LIN {X 0,Y 361.952,Z 273.021,A -85,B 0,C 180,E1 -12972.333,E2 -12972.333} C_VEL
LIN {X 0,Y 361.954,Z 273.018,A -85,B 0,C 180,E1 -12974.621,E2 -12974.621} C_VEL
LIN {X 0,Y 361.95,Z 273.019,A -85,B 0,C 180,E1 -12978.1,E2 -12978.1} C_VEL
LIN {X 0,Y 361.885,Z 273.022,A -85,B 0,C 180,E1 -12981.653,E2 -12981.653} C_VEL
LIN {X 0,Y 361.922,Z 273.026,A -85,B 0,C 180,E1 -12985.29,E2 -12985.29} C_VEL
LIN {X 0,Y 361.916,Z 273.017,A -85,B 0,C 180,E1 -12987.778,E2 -12987.778} C_VEL
LIN {X 0,Y 361.841,Z 273.035,A -85,B 0,C 180,E1 -12991.286,E2 -12991.286} C_VEL
LIN {X 0,Y 361.849,Z 272.995,A -85,B 0,C 180,E1 -12994.281,E2 -12994.281} C_VEL
LIN {X 0,Y 361.86,Z 273.028,A -85,B 0,C 180,E1 -12997.224,E2 -12997.224} C_VEL
LIN {X 0,Y 361.831,Z 273.03,A -85,B 0,C 180,E1 -13000.756,E2 -13000.756} C_VEL
LIN {X 0,Y 361.842,Z 273.033,A -85,B 0,C 180,E1 -13004.365,E2 -13004.365} C_VEL
LIN {X 0,Y 361.88,Z 273.014,A -85,B 0,C 180,E1 -13007.561,E2 -13007.561} C_VEL
LIN {X 0,Y 361.872,Z 273.035,A -85,B 0,C 180,E1 -13010.973,E2 -13010.973} C_VEL
LIN {X 0,Y 361.872,Z 273.035,A -85,B 0,C 180,E1 -13014.656,E2 -13014.656} C_VEL
LIN {X 0,Y 361.866,Z 273.12,A -85,B 0,C 180,E1 -13017.718,E2 -13017.718} C_VEL
LIN {X 0,Y 364.625,Z 284.445,A -85,B 0,C 180,E1 -13020.757,E2 -13020.757} C_VEL
LIN {X 0,Y 366.783,Z 294.302,A -85,B 0,C 180,E1 -13023.166,E2 -13023.166} C_VEL
LIN {X 0,Y 369.556,Z 302.023,A -85,B 0,C 180,E1 -13023.576,E2 -13023.576} C_VEL
LIN {X 0,Y 374.934,Z 329.513,A -85,B 0,C 180,E1 -13024.555,E2 -13024.555} C_VEL
LIN {X 0,Y 373.046,Z 425.138,A -85,B 0,C 180,E1 -13026.401,E2 -13026.401} C_VEL
LIN {X 0,Y 372.477,Z 438.942,A -85,B 0,C 180,E1 -13026.768,E2 -13026.768} C_VEL
LIN {X 0,Y 371.561,Z 452.604,A -85,B 0,C 180,E1 -13027.333,E2 -13027.333} C_VEL
LIN {X 0,Y 370.455,Z 465.982,A -85,B 0,C 180,E1 -13028.106,E2 -13028.106} C_VEL
LIN {X 0,Y 369.2,Z 479.198,A -85,B 0,C 180,E1 -13029.112,E2 -13029.112} C_VEL
LIN {X 0,Y 367.718,Z 491.74,A -85,B 0,C 180,E1 -13030.315,E2 -13030.315} C_VEL
LIN {X 0,Y 366.376,Z 502.198,A -85,B 0,C 180,E1 -13031.548,E2 -13031.548} C_VEL
LIN {X 0,Y 365.092,Z 511.93,A -85,B 0,C 180,E1 -13032.929,E2 -13032.929} C_VEL
LIN {X 0,Y 363.782,Z 521.814,A -85,B 0,C 180,E1 -13034.624,E2 -13034.624} C_VEL
LIN {X 0,Y 362.74,Z 529.741,A -85,B 0,C 180,E1 -13036.271,E2 -13036.271} C_VEL
LIN {X 0,Y 361.767,Z 537.481,A -85,B 0,C 180,E1 -13038.23,E2 -13038.23} C_VEL
LIN {X 0,Y 361.155,Z 542.884,A -85,B 0,C 180,E1 -13039.914,E2 -13039.914} C_VEL
LIN {X 0,Y 360.659,Z 548.569,A -85,B 0,C 180,E1 -13042.16,E2 -13042.16} C_VEL
LIN {X 0,Y 360.407,Z 552.693,A -85,B 0,C 180,E1 -13044.405,E2 -13044.405} C_VEL
LIN {X 0,Y 360.267,Z 555.385,A -85,B 0,C 180,E1 -13046.645,E2 -13046.645} C_VEL
LIN {X 0,Y 360.246,Z 556.718,A -85,B 0,C 180,E1 -13048.882,E2 -13048.882} C_VEL
LIN {X 0,Y 360.246,Z 556.714,A -85,B 0,C 180,E1 -13051.118,E2 -13051.118} C_VEL
LIN {X 0,Y 360.268,Z 555.376,A -85,B 0,C 180,E1 -13053.355,E2 -13053.355} C_VEL
LIN {X 0,Y 360.408,Z 552.678,A -85,B 0,C 180,E1 -13055.595,E2 -13055.595} C_VEL
LIN {X 0,Y 360.659,Z 548.543,A -85,B 0,C 180,E1 -13057.84,E2 -13057.84} C_VEL
LIN {X 0,Y 361.163,Z 542.848,A -85,B 0,C 180,E1 -13060.086,E2 -13060.086} C_VEL
LIN {X 0,Y 361.932,Z 536.429,A -85,B 0,C 180,E1 -13062.049,E2 -13062.049} C_VEL
LIN {X 0,Y 362.885,Z 528.492,A -85,B 0,C 180,E1 -13064.001,E2 -13064.001} C_VEL
LIN {X 0,Y 363.958,Z 520.11,A -85,B 0,C 180,E1 -13065.684,E2 -13065.684} C_VEL
LIN {X 0,Y 365.283,Z 510.065,A -85,B 0,C 180,E1 -13067.35,E2 -13067.35} C_VEL
LIN {X 0,Y 366.763,Z 498.857,A -85,B 0,C 180,E1 -13068.866,E2 -13068.866} C_VEL
LIN {X 0,Y 368.224,Z 487.708,A -85,B 0,C 180,E1 -13070.093,E2 -13070.093} C_VEL
LIN {X 0,Y 369.54,Z 475.56,A -85,B 0,C 180,E1 -13071.182,E2 -13071.182} C_VEL
LIN {X 0,Y 370.771,Z 462.078,A -85,B 0,C 180,E1 -13072.131,E2 -13072.131} C_VEL
LIN {X 0,Y 371.888,Z 447.972,A -85,B 0,C 180,E1 -13072.867,E2 -13072.867} C_VEL
LIN {X 0,Y 372.638,Z 434.166,A -85,B 0,C 180,E1 -13073.369,E2 -13073.369} C_VEL
LIN {X 0,Y 373.32,Z 411.975,A -85,B 0,C 180,E1 -13073.838,E2 -13073.838} C_VEL
LIN {X 0,Y 374.849,Z 329.127,A -85,B 0,C 180,E1 -13075.444,E2 -13075.444} C_VEL
LIN {X 0,Y 369.224,Z 300.604,A -85,B 0,C 180,E1 -13076.464,E2 -13076.464} C_VEL
LIN {X 0,Y 366.745,Z 294.208,A -85,B 0,C 180,E1 -13076.829,E2 -13076.829} C_VEL
LIN {X 0,Y 364.591,Z 284.391,A -85,B 0,C 180,E1 -13079.241,E2 -13079.241} C_VEL
LIN {X 0,Y 361.892,Z 273.253,A -85,B 0,C 180,E1 -13082.197,E2 -13082.197} C_VEL
LIN {X 0,Y 361.852,Z 273.028,A -85,B 0,C 180,E1 -13084.28,E2 -13084.28} C_VEL
LIN {X 0,Y 361.861,Z 273.02,A -85,B 0,C 180,E1 -13087.222,E2 -13087.222} C_VEL
LIN {X 0,Y 361.832,Z 273.02,A -85,B 0,C 180,E1 -13090.755,E2 -13090.755} C_VEL
LIN {X 0,Y 361.816,Z 273.043,A -85,B 0,C 180,E1 -13094.368,E2 -13094.368} C_VEL
LIN {X 0,Y 361.833,Z 273.038,A -85,B 0,C 180,E1 -13097.567,E2 -13097.567} C_VEL
LIN {X 0,Y 361.867,Z 273.034,A -85,B 0,C 180,E1 -13100.973,E2 -13100.973} C_VEL
LIN {X 0,Y 361.87,Z 272.997,A -85,B 0,C 180,E1 -13104.655,E2 -13104.655} C_VEL
LIN {X 0,Y 361.833,Z 273.03,A -85,B 0,C 180,E1 -13108.37,E2 -13108.37} C_VEL
LIN {X 0,Y 361.897,Z 273.027,A -85,B 0,C 180,E1 -13110.955,E2 -13110.955} C_VEL
LIN {X 0,Y 361.949,Z 273.015,A -85,B 0,C 180,E1 -13113.475,E2 -13113.475} C_VEL
LIN {X 0,Y 361.884,Z 273.023,A -85,B 0,C 180,E1 -13117.144,E2 -13117.144} C_VEL
LIN {X 0,Y 361.905,Z 273.028,A -85,B 0,C 180,E1 -13120.723,E2 -13120.723} C_VEL
LIN {X 0,Y 361.926,Z 273.015,A -85,B 0,C 180,E1 -13123.066,E2 -13123.066} C_VEL
LIN {X 0,Y 361.992,Z 273.017,A -85,B 0,C 180,E1 -13126.528,E2 -13126.528} C_VEL
LIN {X 0,Y 362.024,Z 273.001,A -85,B 0,C 180,E1 -13129.938,E2 -13129.938} C_VEL
LIN {X 0,Y 362.144,Z 272.999,A -85,B 0,C 180,E1 -13132.192,E2 -13132.192} C_VEL
LIN {X 0,Y 362.111,Z 272.996,A -85,B 0,C 180,E1 -13134.431,E2 -13134.431} C_VEL
LIN {X 0,Y 362.275,Z 272.979,A -85,B 0,C 180,E1 -13137.776,E2 -13137.776} C_VEL
LIN {X 0,Y 362.42,Z 272.962,A -85,B 0,C 180,E1 -13140,E2 -13140} C_VEL
LIN {X 0,Y 362.276,Z 272.964,A -85,B 0,C 180,E1 -13142.224,E2 -13142.224} C_VEL
LIN {X 0,Y 362.156,Z 272.996,A -85,B 0,C 180,E1 -13146.687,E2 -13146.687} C_VEL
LIN {X 0,Y 362.024,Z 273.008,A -85,B 0,C 180,E1 -13150.062,E2 -13150.062} C_VEL
LIN {X 0,Y 361.991,Z 273.008,A -85,B 0,C 180,E1 -13153.899,E2 -13153.899} C_VEL
LIN {X 0,Y 361.961,Z 273.021,A -85,B 0,C 180,E1 -13157.939,E2 -13157.939} C_VEL
LIN {X 0,Y 361.886,Z 273.024,A -85,B 0,C 180,E1 -13161.653,E2 -13161.653} C_VEL
LIN {X 0,Y 361.923,Z 273.018,A -85,B 0,C 180,E1 -13165.291,E2 -13165.291} C_VEL
LIN {X 0,Y 361.917,Z 273.025,A -85,B 0,C 180,E1 -13167.778,E2 -13167.778} C_VEL
LIN {X 0,Y 361.842,Z 273.019,A -85,B 0,C 180,E1 -13171.286,E2 -13171.286} C_VEL
LIN {X 0,Y 361.85,Z 272.997,A -85,B 0,C 180,E1 -13174.281,E2 -13174.281} C_VEL
LIN {X 0,Y 361.868,Z 273.036,A -85,B 0,C 180,E1 -13177.225,E2 -13177.225} C_VEL
LIN {X 0,Y 361.852,Z 273.006,A -85,B 0,C 180,E1 -13180.76,E2 -13180.76} C_VEL
LIN {X 0,Y 361.832,Z 273.037,A -85,B 0,C 180,E1 -13184.367,E2 -13184.367} C_VEL
LIN {X 0,Y 361.834,Z 273.015,A -85,B 0,C 180,E1 -13187.569,E2 -13187.569} C_VEL
LIN {X 0,Y 361.868,Z 273.03,A -85,B 0,C 180,E1 -13190.974,E2 -13190.974} C_VEL
LIN {X 0,Y 361.873,Z 273.032,A -85,B 0,C 180,E1 -13194.656,E2 -13194.656} C_VEL
LIN {X 0,Y 361.837,Z 273.032,A -85,B 0,C 180,E1 -13198.371,E2 -13198.371} C_VEL
LIN {X 0,Y 361.901,Z 273.139,A -85,B 0,C 180,E1 -13199.064,E2 -13199.064} C_VEL
LIN {X 0,Y 364.583,Z 284.299,A -85,B 0,C 180,E1 -13202.131,E2 -13202.131} C_VEL
LIN {X 0,Y 365.464,Z 288.404,A -85,B 0,C 180,E1 -13203.13,E2 -13203.13} C_VEL
LIN {X 0,Y 371.55,Z 303.667,A -85,B 0,C 180,E1 -13203.956,E2 -13203.956} C_VEL
LIN {X 0,Y 375.122,Z 322.173,A -85,B 0,C 180,E1 -13204.608,E2 -13204.608} C_VEL
LIN {X 0,Y 373.223,Z 410.537,A -85,B 0,C 180,E1 -13206.303,E2 -13206.303} C_VEL
LIN {X 0,Y 372.705,Z 428.632,A -85,B 0,C 180,E1 -13206.709,E2 -13206.709} C_VEL
LIN {X 0,Y 371.91,Z 442.893,A -85,B 0,C 180,E1 -13207.245,E2 -13207.245} C_VEL
LIN {X 0,Y 370.856,Z 457.001,A -85,B 0,C 180,E1 -13208.008,E2 -13208.008} C_VEL
LIN {X 0,Y 369.689,Z 470.266,A -85,B 0,C 180,E1 -13208.972,E2 -13208.972} C_VEL
LIN {X 0,Y 368.352,Z 482.146,A -85,B 0,C 180,E1 -13210.06,E2 -13210.06} C_VEL
LIN {X 0,Y 366.843,Z 494.177,A -85,B 0,C 180,E1 -13211.428,E2 -13211.428} C_VEL
LIN {X 0,Y 365.427,Z 505.023,A -85,B 0,C 180,E1 -13212.945,E2 -13212.945} C_VEL
LIN {X 0,Y 363.998,Z 515.188,A -85,B 0,C 180,E1 -13214.683,E2 -13214.683} C_VEL
LIN {X 0,Y 362.971,Z 524.109,A -85,B 0,C 180,E1 -13216.565,E2 -13216.565} C_VEL
LIN {X 0,Y 362.003,Z 530.634,A -85,B 0,C 180,E1 -13218.238,E2 -13218.238} C_VEL
LIN {X 0,Y 361.393,Z 536.049,A -85,B 0,C 180,E1 -13219.92,E2 -13219.92} C_VEL
LIN {X 0,Y 360.776,Z 541.742,A -85,B 0,C 180,E1 -13222.163,E2 -13222.163} C_VEL
LIN {X 0,Y 360.623,Z 544.719,A -85,B 0,C 180,E1 -13223.677,E2 -13223.677} C_VEL
LIN {X 0,Y 360.423,Z 547.405,A -85,B 0,C 180,E1 -13225.527,E2 -13225.527} C_VEL
LIN {X 0,Y 360.263,Z 549.43,A -85,B 0,C 180,E1 -13227.764,E2 -13227.764} C_VEL
LIN {X 0,Y 360.274,Z 550.124,A -85,B 0,C 180,E1 -13230,E2 -13230} C_VEL
LIN {X 0,Y 360.263,Z 549.497,A -85,B 0,C 180,E1 -13232.236,E2 -13232.236} C_VEL
LIN {X 0,Y 360.423,Z 547.532,A -85,B 0,C 180,E1 -13234.473,E2 -13234.473} C_VEL
LIN {X 0,Y 360.655,Z 544.185,A -85,B 0,C 180,E1 -13236.714,E2 -13236.714} C_VEL
LIN {X 0,Y 361.032,Z 539.358,A -85,B 0,C 180,E1 -13238.959,E2 -13238.959} C_VEL
LIN {X 0,Y 361.73,Z 532.895,A -85,B 0,C 180,E1 -13241.203,E2 -13241.203} C_VEL
LIN {X 0,Y 362.715,Z 525.696,A -85,B 0,C 180,E1 -13243.159,E2 -13243.159} C_VEL
LIN {X 0,Y 363.758,Z 517.473,A -85,B 0,C 180,E1 -13244.977,E2 -13244.977} C_VEL
LIN {X 0,Y 364.828,Z 509.096,A -85,B 0,C 180,E1 -13246.507,E2 -13246.507} C_VEL
LIN {X 0,Y 366.341,Z 498.123,A -85,B 0,C 180,E1 -13248.164,E2 -13248.164} C_VEL
LIN {X 0,Y 367.661,Z 488.275,A -85,B 0,C 180,E1 -13249.38,E2 -13249.38} C_VEL
LIN {X 0,Y 367.626,Z 483.577,A -85,B 0,C 180,E1 -13249.941,E2 -13249.941} C_VEL
LIN {X 0,Y 365.814,Z 475.828,A -85,B 0,C 180,E1 -13250.871,E2 -13250.871} C_VEL
LIN {X 0,Y 363.955,Z 467.722,A -85,B 0,C 180,E1 -13251.719,E2 -13251.719} C_VEL
LIN {X 0,Y 363.828,Z 462.47,A -85,B 0,C 180,E1 -13252.144,E2 -13252.144} C_VEL
LIN {X 0,Y 365.032,Z 448.328,A -85,B 0,C 180,E1 -13253.021,E2 -13253.021} C_VEL
LIN {X 0,Y 365.932,Z 434.613,A -85,B 0,C 180,E1 -13253.635,E2 -13253.635} C_VEL
LIN {X 0,Y 366.616,Z 420.613,A -85,B 0,C 180,E1 -13254.038,E2 -13254.038} C_VEL
LIN {X 0,Y 368.716,Z 323.276,A -85,B 0,C 180,E1 -13255.95,E2 -13255.95} C_VEL
LIN {X 0,Y 365.307,Z 305.617,A -85,B 0,C 180,E1 -13256.591,E2 -13256.591} C_VEL
LIN {X 0,Y 358.198,Z 288.358,A -85,B 0,C 180,E1 -13257.582,E2 -13257.582} C_VEL
LIN {X 0,Y 355.906,Z 278.366,A -85,B 0,C 180,E1 -13260.247,E2 -13260.247} C_VEL
LIN {X 0,Y 354.815,Z 273.973,A -85,B 0,C 180,E1 -13261.57,E2 -13261.57} C_VEL
LIN {X 0,Y 354.81,Z 273.909,A -85,B 0,C 180,E1 -13265.058,E2 -13265.058} C_VEL
LIN {X 0,Y 354.804,Z 273.901,A -85,B 0,C 180,E1 -13267.882,E2 -13267.882} C_VEL
LIN {X 0,Y 354.786,Z 273.905,A -85,B 0,C 180,E1 -13271.171,E2 -13271.171} C_VEL
LIN {X 0,Y 354.787,Z 273.914,A -85,B 0,C 180,E1 -13274.51,E2 -13274.51} C_VEL
LIN {X 0,Y 354.796,Z 273.888,A -85,B 0,C 180,E1 -13277.663,E2 -13277.663} C_VEL
LIN {X 0,Y 354.815,Z 273.904,A -85,B 0,C 180,E1 -13280.666,E2 -13280.666} C_VEL
LIN {X 0,Y 354.817,Z 273.902,A -85,B 0,C 180,E1 -13284.3,E2 -13284.3} C_VEL
LIN {X 0,Y 354.782,Z 273.881,A -85,B 0,C 180,E1 -13287.666,E2 -13287.666} C_VEL
LIN {X 0,Y 354.863,Z 273.906,A -85,B 0,C 180,E1 -13290.621,E2 -13290.621} C_VEL
LIN {X 0,Y 354.893,Z 273.89,A -85,B 0,C 180,E1 -13294.172,E2 -13294.172} C_VEL
LIN {X 0,Y 354.828,Z 273.905,A -85,B 0,C 180,E1 -13297.893,E2 -13297.893} C_VEL
LIN {X 0,Y 354.916,Z 273.898,A -85,B 0,C 180,E1 -13301.891,E2 -13301.891} C_VEL
LIN {X 0,Y 354.935,Z 273.886,A -85,B 0,C 180,E1 -13305.981,E2 -13305.981} C_VEL
LIN {X 0,Y 354.971,Z 273.886,A -85,B 0,C 180,E1 -13309.736,E2 -13309.736} C_VEL
LIN {X 0,Y 355.12,Z 273.873,A -85,B 0,C 180,E1 -13313.18,E2 -13313.18} C_VEL
LIN {X 0,Y 355.238,Z 273.84,A -85,B 0,C 180,E1 -13317.732,E2 -13317.732} C_VEL
LIN {X 0,Y 355.391,Z 273.837,A -85,B 0,C 180,E1 -13320,E2 -13320} C_VEL
LIN {X 0,Y 355.238,Z 273.855,A -85,B 0,C 180,E1 -13322.268,E2 -13322.268} C_VEL
LIN {X 0,Y 355.13,Z 273.873,A -85,B 0,C 180,E1 -13326.819,E2 -13326.819} C_VEL
LIN {X 0,Y 355.007,Z 273.878,A -85,B 0,C 180,E1 -13329.112,E2 -13329.112} C_VEL
LIN {X 0,Y 354.913,Z 273.901,A -85,B 0,C 180,E1 -13332.581,E2 -13332.581} C_VEL
LIN {X 0,Y 354.882,Z 273.891,A -85,B 0,C 180,E1 -13336.096,E2 -13336.096} C_VEL
LIN {X 0,Y 354.896,Z 273.903,A -85,B 0,C 180,E1 -13338.472,E2 -13338.472} C_VEL
LIN {X 0,Y 354.828,Z 273.899,A -85,B 0,C 180,E1 -13342.106,E2 -13342.106} C_VEL
LIN {X 0,Y 354.893,Z 273.901,A -85,B 0,C 180,E1 -13345.828,E2 -13345.828} C_VEL
LIN {X 0,Y 354.848,Z 273.909,A -85,B 0,C 180,E1 -13349.679,E2 -13349.679} C_VEL
LIN {X 0,Y 354.801,Z 273.875,A -85,B 0,C 180,E1 -13353.703,E2 -13353.703} C_VEL
LIN {X 0,Y 354.793,Z 273.896,A -85,B 0,C 180,E1 -13356.46,E2 -13356.46} C_VEL
LIN {X 0,Y 354.819,Z 273.911,A -85,B 0,C 180,E1 -13359.424,E2 -13359.424} C_VEL
LIN {X 0,Y 354.786,Z 273.915,A -85,B 0,C 180,E1 -13362.868,E2 -13362.868} C_VEL
LIN {X 0,Y 354.837,Z 273.908,A -85,B 0,C 180,E1 -13366.116,E2 -13366.116} C_VEL
LIN {X 0,Y 354.853,Z 273.889,A -85,B 0,C 180,E1 -13369.189,E2 -13369.189} C_VEL
LIN {X 0,Y 354.806,Z 273.899,A -85,B 0,C 180,E1 -13372.403,E2 -13372.403} C_VEL
LIN {X 0,Y 354.81,Z 273.915,A -85,B 0,C 180,E1 -13374.942,E2 -13374.942} C_VEL
LIN {X 0,Y 354.846,Z 274.024,A -85,B 0,C 180,E1 -13377.253,E2 -13377.253} C_VEL
LIN {X 0,Y 357.781,Z 286.229,A -85,B 0,C 180,E1 -13380.589,E2 -13380.589} C_VEL
LIN {X 0,Y 359.57,Z 294.104,A -85,B 0,C 180,E1 -13382.57,E2 -13382.57} C_VEL
LIN {X 0,Y 363.378,Z 304.123,A -85,B 0,C 180,E1 -13383.137,E2 -13383.137} C_VEL
LIN {X 0,Y 368.52,Z 330.505,A -85,B 0,C 180,E1 -13384.102,E2 -13384.102} C_VEL
LIN {X 0,Y 366.561,Z 425.089,A -85,B 0,C 180,E1 -13385.958,E2 -13385.958} C_VEL
LIN {X 0,Y 365.955,Z 438.886,A -85,B 0,C 180,E1 -13386.329,E2 -13386.329} C_VEL
LIN {X 0,Y 365.028,Z 452.545,A -85,B 0,C 180,E1 -13386.904,E2 -13386.904} C_VEL
LIN {X 0,Y 363.867,Z 465.921,A -85,B 0,C 180,E1 -13387.688,E2 -13387.688} C_VEL
LIN {X 0,Y 362.68,Z 477.912,A -85,B 0,C 180,E1 -13388.603,E2 -13388.603} C_VEL
LIN {X 0,Y 361.209,Z 490.384,A -85,B 0,C 180,E1 -13389.797,E2 -13389.797} C_VEL
LIN {X 0,Y 359.588,Z 502.134,A -85,B 0,C 180,E1 -13391.187,E2 -13391.187} C_VEL
LIN {X 0,Y 358.278,Z 511.866,A -85,B 0,C 180,E1 -13392.594,E2 -13392.594} C_VEL
LIN {X 0,Y 356.897,Z 521.749,A -85,B 0,C 180,E1 -13394.32,E2 -13394.32} C_VEL
LIN {X 0,Y 355.646,Z 530.909,A -85,B 0,C 180,E1 -13396.283,E2 -13396.283} C_VEL
LIN {X 0,Y 354.798,Z 537.416,A -85,B 0,C 180,E1 -13397.996,E2 -13397.996} C_VEL
LIN {X 0,Y 354.138,Z 542.818,A -85,B 0,C 180,E1 -13399.712,E2 -13399.712} C_VEL
LIN {X 0,Y 353.602,Z 548.503,A -85,B 0,C 180,E1 -13402.003,E2 -13402.003} C_VEL
LIN {X 0,Y 353.329,Z 552.627,A -85,B 0,C 180,E1 -13404.292,E2 -13404.292} C_VEL
LIN {X 0,Y 353.191,Z 555.319,A -85,B 0,C 180,E1 -13406.578,E2 -13406.578} C_VEL
LIN {X 0,Y 353.146,Z 556.651,A -85,B 0,C 180,E1 -13408.86,E2 -13408.86} C_VEL
LIN {X 0,Y 353.146,Z 556.648,A -85,B 0,C 180,E1 -13411.14,E2 -13411.14} C_VEL
LIN {X 0,Y 353.191,Z 555.31,A -85,B 0,C 180,E1 -13413.422,E2 -13413.422} C_VEL
LIN {X 0,Y 353.329,Z 552.611,A -85,B 0,C 180,E1 -13415.708,E2 -13415.708} C_VEL
LIN {X 0,Y 353.602,Z 548.475,A -85,B 0,C 180,E1 -13417.997,E2 -13417.997} C_VEL
LIN {X 0,Y 354.144,Z 542.78,A -85,B 0,C 180,E1 -13420.288,E2 -13420.288} C_VEL
LIN {X 0,Y 354.96,Z 536.361,A -85,B 0,C 180,E1 -13422.289,E2 -13422.289} C_VEL
LIN {X 0,Y 355.924,Z 528.696,A -85,B 0,C 180,E1 -13424.216,E2 -13424.216} C_VEL
LIN {X 0,Y 357.072,Z 520.041,A -85,B 0,C 180,E1 -13425.995,E2 -13425.995} C_VEL
LIN {X 0,Y 358.484,Z 509.996,A -85,B 0,C 180,E1 -13427.69,E2 -13427.69} C_VEL
LIN {X 0,Y 360.048,Z 498.787,A -85,B 0,C 180,E1 -13429.232,E2 -13429.232} C_VEL
LIN {X 0,Y 361.704,Z 486.351,A -85,B 0,C 180,E1 -13430.605,E2 -13430.605} C_VEL
LIN {X 0,Y 363.131,Z 473.38,A -85,B 0,C 180,E1 -13431.753,E2 -13431.753} C_VEL
LIN {X 0,Y 364.32,Z 460.986,A -85,B 0,C 180,E1 -13432.612,E2 -13432.612} C_VEL
LIN {X 0,Y 365.423,Z 447.135,A -85,B 0,C 180,E1 -13433.332,E2 -13433.332} C_VEL
LIN {X 0,Y 366.189,Z 432.947,A -85,B 0,C 180,E1 -13433.843,E2 -13433.843} C_VEL
LIN {X 0,Y 367.019,Z 402.941,A -85,B 0,C 180,E1 -13434.462,E2 -13434.462} C_VEL
LIN {X 0,Y 368.44,Z 330.261,A -85,B 0,C 180,E1 -13435.894,E2 -13435.894} C_VEL
LIN {X 0,Y 363.186,Z 303.268,A -85,B 0,C 180,E1 -13436.879,E2 -13436.879} C_VEL
LIN {X 0,Y 359.527,Z 294.085,A -85,B 0,C 180,E1 -13437.418,E2 -13437.418} C_VEL
LIN {X 0,Y 356.951,Z 282.742,A -85,B 0,C 180,E1 -13440.312,E2 -13440.312} C_VEL
LIN {X 0,Y 354.846,Z 273.997,A -85,B 0,C 180,E1 -13442.747,E2 -13442.747} C_VEL
LIN {X 0,Y 354.795,Z 273.902,A -85,B 0,C 180,E1 -13446.459,E2 -13446.459} C_VEL
LIN {X 0,Y 354.821,Z 273.912,A -85,B 0,C 180,E1 -13449.423,E2 -13449.423} C_VEL
LIN {X 0,Y 354.785,Z 273.904,A -85,B 0,C 180,E1 -13452.867,E2 -13452.867} C_VEL
LIN {X 0,Y 354.764,Z 273.914,A -85,B 0,C 180,E1 -13456.103,E2 -13456.103} C_VEL
LIN {X 0,Y 354.784,Z 273.907,A -85,B 0,C 180,E1 -13459.178,E2 -13459.178} C_VEL
LIN {X 0,Y 354.804,Z 273.909,A -85,B 0,C 180,E1 -13462.402,E2 -13462.402} C_VEL
LIN {X 0,Y 354.807,Z 273.872,A -85,B 0,C 180,E1 -13464.94,E2 -13464.94} C_VEL
LIN {X 0,Y 354.789,Z 273.907,A -85,B 0,C 180,E1 -13468.404,E2 -13468.404} C_VEL
LIN {X 0,Y 354.848,Z 273.902,A -85,B 0,C 180,E1 -13471.619,E2 -13471.619} C_VEL
LIN {X 0,Y 354.894,Z 273.902,A -85,B 0,C 180,E1 -13474.172,E2 -13474.172} C_VEL
LIN {X 0,Y 354.828,Z 273.899,A -85,B 0,C 180,E1 -13477.894,E2 -13477.894} C_VEL
LIN {X 0,Y 354.916,Z 273.894,A -85,B 0,C 180,E1 -13481.891,E2 -13481.891} C_VEL
LIN {X 0,Y 354.936,Z 273.9,A -85,B 0,C 180,E1 -13485.981,E2 -13485.981} C_VEL
LIN {X 0,Y 354.971,Z 273.878,A -85,B 0,C 180,E1 -13489.736,E2 -13489.736} C_VEL
LIN {X 0,Y 355.107,Z 273.876,A -85,B 0,C 180,E1 -13492.037,E2 -13492.037} C_VEL
LIN {X 0,Y 355.085,Z 273.871,A -85,B 0,C 180,E1 -13494.321,E2 -13494.321} C_VEL
LIN {X 0,Y 355.239,Z 273.854,A -85,B 0,C 180,E1 -13497.732,E2 -13497.732} C_VEL
LIN {X 0,Y 355.39,Z 273.838,A -85,B 0,C 180,E1 -13500,E2 -13500} C_VEL
LIN {X 0,Y 355.239,Z 273.84,A -85,B 0,C 180,E1 -13502.268,E2 -13502.268} C_VEL
LIN {X 0,Y 355.12,Z 273.873,A -85,B 0,C 180,E1 -13506.82,E2 -13506.82} C_VEL
LIN {X 0,Y 354.971,Z 273.886,A -85,B 0,C 180,E1 -13510.264,E2 -13510.264} C_VEL
LIN {X 0,Y 354.936,Z 273.886,A -85,B 0,C 180,E1 -13514.019,E2 -13514.019} C_VEL
LIN {X 0,Y 354.916,Z 273.898,A -85,B 0,C 180,E1 -13518.109,E2 -13518.109} C_VEL
LIN {X 0,Y 354.829,Z 273.905,A -85,B 0,C 180,E1 -13522.107,E2 -13522.107} C_VEL
LIN {X 0,Y 354.894,Z 273.89,A -85,B 0,C 180,E1 -13525.828,E2 -13525.828} C_VEL
LIN {X 0,Y 354.85,Z 273.905,A -85,B 0,C 180,E1 -13529.679,E2 -13529.679} C_VEL
LIN {X 0,Y 354.802,Z 273.87,A -85,B 0,C 180,E1 -13533.703,E2 -13533.703} C_VEL
LIN {X 0,Y 354.798,Z 273.907,A -85,B 0,C 180,E1 -13536.46,E2 -13536.46} C_VEL
LIN {X 0,Y 354.821,Z 273.902,A -85,B 0,C 180,E1 -13539.424,E2 -13539.424} C_VEL
LIN {X 0,Y 354.788,Z 273.893,A -85,B 0,C 180,E1 -13542.868,E2 -13542.868} C_VEL
LIN {X 0,Y 354.774,Z 273.911,A -85,B 0,C 180,E1 -13546.106,E2 -13546.106} C_VEL
LIN {X 0,Y 354.786,Z 273.908,A -85,B 0,C 180,E1 -13549.18,E2 -13549.18} C_VEL
LIN {X 0,Y 354.806,Z 273.9,A -85,B 0,C 180,E1 -13552.403,E2 -13552.403} C_VEL
LIN {X 0,Y 354.811,Z 273.909,A -85,B 0,C 180,E1 -13554.941,E2 -13554.941} C_VEL
LIN {X 0,Y 354.833,Z 273.986,A -85,B 0,C 180,E1 -13558.567,E2 -13558.567} C_VEL
LIN {X 0,Y 357.337,Z 284.373,A -85,B 0,C 180,E1 -13561.515,E2 -13561.515} C_VEL
LIN {X 0,Y 358.247,Z 288.417,A -85,B 0,C 180,E1 -13562.537,E2 -13562.537} C_VEL
LIN {X 0,Y 365.452,Z 306.188,A -85,B 0,C 180,E1 -13563.54,E2 -13563.54} C_VEL
LIN {X 0,Y 368.722,Z 323.447,A -85,B 0,C 180,E1 -13564.16,E2 -13564.16} C_VEL
LIN {X 0,Y 366.413,Z 425.293,A -85,B 0,C 180,E1 -13566.173,E2 -13566.173} C_VEL
LIN {X 0,Y 365.636,Z 439.165,A -85,B 0,C 180,E1 -13566.645,E2 -13566.645} C_VEL
LIN {X 0,Y 364.635,Z 452.755,A -85,B 0,C 180,E1 -13567.327,E2 -13567.327} C_VEL
LIN {X 0,Y 363.445,Z 466.194,A -85,B 0,C 180,E1 -13568.24,E2 -13568.24} C_VEL
LIN {X 0,Y 362.045,Z 479.427,A -85,B 0,C 180,E1 -13569.4,E2 -13569.4} C_VEL
LIN {X 0,Y 360.556,Z 490.881,A -85,B 0,C 180,E1 -13570.649,E2 -13570.649} C_VEL
LIN {X 0,Y 359.147,Z 501.393,A -85,B 0,C 180,E1 -13572.049,E2 -13572.049} C_VEL
LIN {X 0,Y 357.609,Z 511.831,A -85,B 0,C 180,E1 -13573.737,E2 -13573.737} C_VEL
LIN {X 0,Y 356.449,Z 520.439,A -85,B 0,C 180,E1 -13575.441,E2 -13575.441} C_VEL
LIN {X 0,Y 355.53,Z 527.591,A -85,B 0,C 180,E1 -13577.151,E2 -13577.151} C_VEL
LIN {X 0,Y 354.561,Z 534.44,A -85,B 0,C 180,E1 -13579.146,E2 -13579.146} C_VEL
LIN {X 0,Y 353.995,Z 539.167,A -85,B 0,C 180,E1 -13580.861,E2 -13580.861} C_VEL
LIN {X 0,Y 353.59,Z 544.064,A -85,B 0,C 180,E1 -13583.151,E2 -13583.151} C_VEL
LIN {X 0,Y 353.338,Z 547.472,A -85,B 0,C 180,E1 -13585.437,E2 -13585.437} C_VEL
LIN {X 0,Y 353.172,Z 549.497,A -85,B 0,C 180,E1 -13587.719,E2 -13587.719} C_VEL
LIN {X 0,Y 353.175,Z 550.191,A -85,B 0,C 180,E1 -13590,E2 -13590} C_VEL
LIN {X 0,Y 353.171,Z 549.563,A -85,B 0,C 180,E1 -13592.281,E2 -13592.281} C_VEL
LIN {X 0,Y 353.338,Z 547.598,A -85,B 0,C 180,E1 -13594.563,E2 -13594.563} C_VEL
LIN {X 0,Y 353.59,Z 544.251,A -85,B 0,C 180,E1 -13596.849,E2 -13596.849} C_VEL
LIN {X 0,Y 353.983,Z 539.424,A -85,B 0,C 180,E1 -13599.139,E2 -13599.139} C_VEL
LIN {X 0,Y 354.722,Z 532.96,A -85,B 0,C 180,E1 -13601.427,E2 -13601.427} C_VEL
LIN {X 0,Y 355.782,Z 525.761,A -85,B 0,C 180,E1 -13603.421,E2 -13603.421} C_VEL
LIN {X 0,Y 356.77,Z 518.134,A -85,B 0,C 180,E1 -13605.148,E2 -13605.148} C_VEL
LIN {X 0,Y 357.997,Z 509.16,A -85,B 0,C 180,E1 -13606.831,E2 -13606.831} C_VEL
LIN {X 0,Y 359.556,Z 498.187,A -85,B 0,C 180,E1 -13608.519,E2 -13608.519} C_VEL
LIN {X 0,Y 361.129,Z 486.994,A -85,B 0,C 180,E1 -13609.911,E2 -13609.911} C_VEL
LIN {X 0,Y 362.659,Z 474.609,A -85,B 0,C 180,E1 -13611.157,E2 -13611.157} C_VEL
LIN {X 0,Y 363.828,Z 462.47,A -85,B 0,C 180,E1 -13612.144,E2 -13612.144} C_VEL
LIN {X 0,Y 363.75,Z 457.116,A -85,B 0,C 180,E1 -13612.548,E2 -13612.548} C_VEL
LIN {X 0,Y 361.716,Z 448.423,A -85,B 0,C 180,E1 -13613.24,E2 -13613.24} C_VEL
LIN {X 0,Y 359.73,Z 439.54,A -85,B 0,C 180,E1 -13613.854,E2 -13613.854} C_VEL
LIN {X 0,Y 359.526,Z 433.901,A -85,B 0,C 180,E1 -13614.115,E2 -13614.115} C_VEL
LIN {X 0,Y 360.155,Z 420.658,A -85,B 0,C 180,E1 -13614.498,E2 -13614.498} C_VEL
LIN {X 0,Y 362.327,Z 324.486,A -85,B 0,C 180,E1 -13616.417,E2 -13616.417} C_VEL
LIN {X 0,Y 359.741,Z 310.295,A -85,B 0,C 180,E1 -13616.933,E2 -13616.933} C_VEL
LIN {X 0,Y 358.312,Z 305.765,A -85,B 0,C 180,E1 -13617.15,E2 -13617.15} C_VEL
LIN {X 0,Y 351.028,Z 288.415,A -85,B 0,C 180,E1 -13618.196,E2 -13618.196} C_VEL
LIN {X 0,Y 348.68,Z 278.488,A -85,B 0,C 180,E1 -13620.928,E2 -13620.928} C_VEL
LIN {X 0,Y 347.758,Z 274.836,A -85,B 0,C 180,E1 -13622.08,E2 -13622.08} C_VEL
LIN {X 0,Y 347.769,Z 274.794,A -85,B 0,C 180,E1 -13626.064,E2 -13626.064} C_VEL
LIN {X 0,Y 347.75,Z 274.785,A -85,B 0,C 180,E1 -13628.792,E2 -13628.792} C_VEL
LIN {X 0,Y 347.748,Z 274.773,A -85,B 0,C 180,E1 -13631.829,E2 -13631.829} C_VEL
LIN {X 0,Y 347.763,Z 274.791,A -85,B 0,C 180,E1 -13635.016,E2 -13635.016} C_VEL
LIN {X 0,Y 347.755,Z 274.759,A -85,B 0,C 180,E1 -13638.395,E2 -13638.395} C_VEL
LIN {X 0,Y 347.771,Z 274.793,A -85,B 0,C 180,E1 -13642.01,E2 -13642.01} C_VEL
LIN {X 0,Y 347.739,Z 274.76,A -85,B 0,C 180,E1 -13645.535,E2 -13645.535} C_VEL
LIN {X 0,Y 347.759,Z 274.785,A -85,B 0,C 180,E1 -13649.653,E2 -13649.653} C_VEL
LIN {X 0,Y 347.847,Z 274.776,A -85,B 0,C 180,E1 -13652.744,E2 -13652.744} C_VEL
LIN {X 0,Y 347.782,Z 274.787,A -85,B 0,C 180,E1 -13656.161,E2 -13656.161} C_VEL
LIN {X 0,Y 347.806,Z 274.775,A -85,B 0,C 180,E1 -13659.909,E2 -13659.909} C_VEL
LIN {X 0,Y 347.859,Z 274.779,A -85,B 0,C 180,E1 -13662.359,E2 -13662.359} C_VEL
LIN {X 0,Y 347.891,Z 274.763,A -85,B 0,C 180,E1 -13665.97,E2 -13665.97} C_VEL
LIN {X 0,Y 347.921,Z 274.764,A -85,B 0,C 180,E1 -13669.525,E2 -13669.525} C_VEL
LIN {X 0,Y 348.086,Z 274.748,A -85,B 0,C 180,E1 -13673.042,E2 -13673.042} C_VEL
LIN {X 0,Y 348.201,Z 274.716,A -85,B 0,C 180,E1 -13677.686,E2 -13677.686} C_VEL
LIN {X 0,Y 348.361,Z 274.713,A -85,B 0,C 180,E1 -13680,E2 -13680} C_VEL
LIN {X 0,Y 348.2,Z 274.73,A -85,B 0,C 180,E1 -13682.313,E2 -13682.313} C_VEL
LIN {X 0,Y 348.098,Z 274.748,A -85,B 0,C 180,E1 -13686.958,E2 -13686.958} C_VEL
LIN {X 0,Y 347.96,Z 274.756,A -85,B 0,C 180,E1 -13689.299,E2 -13689.299} C_VEL
LIN {X 0,Y 347.882,Z 274.776,A -85,B 0,C 180,E1 -13692.84,E2 -13692.84} C_VEL
LIN {X 0,Y 347.831,Z 274.768,A -85,B 0,C 180,E1 -13696.432,E2 -13696.432} C_VEL
LIN {X 0,Y 347.846,Z 274.78,A -85,B 0,C 180,E1 -13698.861,E2 -13698.861} C_VEL
LIN {X 0,Y 347.767,Z 274.779,A -85,B 0,C 180,E1 -13702.58,E2 -13702.58} C_VEL
LIN {X 0,Y 347.806,Z 274.784,A -85,B 0,C 180,E1 -13705.109,E2 -13705.109} C_VEL
LIN {X 0,Y 347.806,Z 274.774,A -85,B 0,C 180,E1 -13707.694,E2 -13707.694} C_VEL
LIN {X 0,Y 347.759,Z 274.791,A -85,B 0,C 180,E1 -13710.347,E2 -13710.347} C_VEL
LIN {X 0,Y 347.739,Z 274.75,A -85,B 0,C 180,E1 -13714.465,E2 -13714.465} C_VEL
LIN {X 0,Y 347.769,Z 274.79,A -85,B 0,C 180,E1 -13717.989,E2 -13717.989} C_VEL
LIN {X 0,Y 347.746,Z 274.793,A -85,B 0,C 180,E1 -13721.831,E2 -13721.831} C_VEL
LIN {X 0,Y 347.793,Z 274.785,A -85,B 0,C 180,E1 -13725.012,E2 -13725.012} C_VEL
LIN {X 0,Y 347.781,Z 274.765,A -85,B 0,C 180,E1 -13728.392,E2 -13728.392} C_VEL
LIN {X 0,Y 347.774,Z 274.779,A -85,B 0,C 180,E1 -13732.011,E2 -13732.011} C_VEL
LIN {X 0,Y 347.742,Z 274.786,A -85,B 0,C 180,E1 -13735.537,E2 -13735.537} C_VEL
LIN {X 0,Y 347.799,Z 274.95,A -85,B 0,C 180,E1 -13736.773,E2 -13736.773} C_VEL
LIN {X 0,Y 350.523,Z 286.159,A -85,B 0,C 180,E1 -13739.918,E2 -13739.918} C_VEL
LIN {X 0,Y 352.332,Z 294.004,A -85,B 0,C 180,E1 -13741.954,E2 -13741.954} C_VEL
LIN {X 0,Y 357.179,Z 306.026,A -85,B 0,C 180,E1 -13742.676,E2 -13742.676} C_VEL
LIN {X 0,Y 362.087,Z 331.302,A -85,B 0,C 180,E1 -13743.625,E2 -13743.625} C_VEL
LIN {X 0,Y 360.25,Z 417.947,A -85,B 0,C 180,E1 -13745.355,E2 -13745.355} C_VEL
LIN {X 0,Y 359.647,Z 435.647,A -85,B 0,C 180,E1 -13745.773,E2 -13745.773} C_VEL
LIN {X 0,Y 358.737,Z 449.687,A -85,B 0,C 180,E1 -13746.322,E2 -13746.322} C_VEL
LIN {X 0,Y 357.547,Z 463.644,A -85,B 0,C 180,E1 -13747.104,E2 -13747.104} C_VEL
LIN {X 0,Y 356.19,Z 476.756,A -85,B 0,C 180,E1 -13748.088,E2 -13748.088} C_VEL
LIN {X 0,Y 354.72,Z 489.029,A -85,B 0,C 180,E1 -13749.259,E2 -13749.259} C_VEL
LIN {X 0,Y 353.003,Z 501,A -85,B 0,C 180,E1 -13750.672,E2 -13750.672} C_VEL
LIN {X 0,Y 351.455,Z 511.801,A -85,B 0,C 180,E1 -13752.245,E2 -13752.245} C_VEL
LIN {X 0,Y 350.039,Z 521.535,A -85,B 0,C 180,E1 -13753.975,E2 -13753.975} C_VEL
LIN {X 0,Y 348.877,Z 529.712,A -85,B 0,C 180,E1 -13755.738,E2 -13755.738} C_VEL
LIN {X 0,Y 347.835,Z 537.351,A -85,B 0,C 180,E1 -13757.752,E2 -13757.752} C_VEL
LIN {X 0,Y 347.108,Z 542.753,A -85,B 0,C 180,E1 -13759.501,E2 -13759.501} C_VEL
LIN {X 0,Y 346.539,Z 548.437,A -85,B 0,C 180,E1 -13761.839,E2 -13761.839} C_VEL
LIN {X 0,Y 346.248,Z 552.56,A -85,B 0,C 180,E1 -13764.175,E2 -13764.175} C_VEL
LIN {X 0,Y 346.117,Z 555.253,A -85,B 0,C 180,E1 -13766.508,E2 -13766.508} C_VEL
LIN {X 0,Y 346.048,Z 556.585,A -85,B 0,C 180,E1 -13768.836,E2 -13768.836} C_VEL
LIN {X 0,Y 346.048,Z 556.581,A -85,B 0,C 180,E1 -13771.164,E2 -13771.164} C_VEL
LIN {X 0,Y 346.117,Z 555.243,A -85,B 0,C 180,E1 -13773.492,E2 -13773.492} C_VEL
LIN {X 0,Y 346.248,Z 552.544,A -85,B 0,C 180,E1 -13775.825,E2 -13775.825} C_VEL
LIN {X 0,Y 346.539,Z 548.407,A -85,B 0,C 180,E1 -13778.161,E2 -13778.161} C_VEL
LIN {X 0,Y 347.113,Z 542.712,A -85,B 0,C 180,E1 -13780.499,E2 -13780.499} C_VEL
LIN {X 0,Y 347.994,Z 536.292,A -85,B 0,C 180,E1 -13782.539,E2 -13782.539} C_VEL
LIN {X 0,Y 349.005,Z 528.641,A -85,B 0,C 180,E1 -13784.5,E2 -13784.5} C_VEL
LIN {X 0,Y 350.218,Z 519.972,A -85,B 0,C 180,E1 -13786.316,E2 -13786.316} C_VEL
LIN {X 0,Y 351.708,Z 509.926,A -85,B 0,C 180,E1 -13788.043,E2 -13788.043} C_VEL
LIN {X 0,Y 353.336,Z 498.717,A -85,B 0,C 180,E1 -13789.612,E2 -13789.612} C_VEL
LIN {X 0,Y 355.041,Z 486.385,A -85,B 0,C 180,E1 -13790.999,E2 -13790.999} C_VEL
LIN {X 0,Y 356.512,Z 473.649,A -85,B 0,C 180,E1 -13792.148,E2 -13792.148} C_VEL
LIN {X 0,Y 357.769,Z 460.8,A -85,B 0,C 180,E1 -13793.057,E2 -13793.057} C_VEL
LIN {X 0,Y 358.963,Z 446.297,A -85,B 0,C 180,E1 -13793.816,E2 -13793.816} C_VEL
LIN {X 0,Y 359.714,Z 432.868,A -85,B 0,C 180,E1 -13794.299,E2 -13794.299} C_VEL
LIN {X 0,Y 360.552,Z 404.644,A -85,B 0,C 180,E1 -13794.892,E2 -13794.892} C_VEL
LIN {X 0,Y 362.042,Z 331.17,A -85,B 0,C 180,E1 -13796.364,E2 -13796.364} C_VEL
LIN {X 0,Y 357.02,Z 305.614,A -85,B 0,C 180,E1 -13797.328,E2 -13797.328} C_VEL
LIN {X 0,Y 352.351,Z 294.099,A -85,B 0,C 180,E1 -13798.014,E2 -13798.014} C_VEL
LIN {X 0,Y 349.543,Z 282.018,A -85,B 0,C 180,E1 -13801.187,E2 -13801.187} C_VEL
LIN {X 0,Y 347.8,Z 274.92,A -85,B 0,C 180,E1 -13803.227,E2 -13803.227} C_VEL
LIN {X 0,Y 347.768,Z 274.781,A -85,B 0,C 180,E1 -13806.064,E2 -13806.064} C_VEL
LIN {X 0,Y 347.749,Z 274.793,A -85,B 0,C 180,E1 -13808.792,E2 -13808.792} C_VEL
LIN {X 0,Y 347.748,Z 274.769,A -85,B 0,C 180,E1 -13811.83,E2 -13811.83} C_VEL
LIN {X 0,Y 347.703,Z 274.796,A -85,B 0,C 180,E1 -13815.026,E2 -13815.026} C_VEL
LIN {X 0,Y 347.746,Z 274.789,A -85,B 0,C 180,E1 -13818.397,E2 -13818.397} C_VEL
LIN {X 0,Y 347.77,Z 274.789,A -85,B 0,C 180,E1 -13822.011,E2 -13822.011} C_VEL
LIN {X 0,Y 347.739,Z 274.749,A -85,B 0,C 180,E1 -13825.536,E2 -13825.536} C_VEL
LIN {X 0,Y 347.759,Z 274.791,A -85,B 0,C 180,E1 -13829.653,E2 -13829.653} C_VEL
LIN {X 0,Y 347.847,Z 274.769,A -85,B 0,C 180,E1 -13832.744,E2 -13832.744} C_VEL
LIN {X 0,Y 347.782,Z 274.784,A -85,B 0,C 180,E1 -13836.162,E2 -13836.162} C_VEL
LIN {X 0,Y 347.808,Z 274.785,A -85,B 0,C 180,E1 -13839.909,E2 -13839.909} C_VEL
LIN {X 0,Y 347.86,Z 274.769,A -85,B 0,C 180,E1 -13842.359,E2 -13842.359} C_VEL
LIN {X 0,Y 347.891,Z 274.777,A -85,B 0,C 180,E1 -13845.971,E2 -13845.971} C_VEL
LIN {X 0,Y 347.921,Z 274.756,A -85,B 0,C 180,E1 -13849.525,E2 -13849.525} C_VEL
LIN {X 0,Y 348.067,Z 274.752,A -85,B 0,C 180,E1 -13851.875,E2 -13851.875} C_VEL
LIN {X 0,Y 348.06,Z 274.747,A -85,B 0,C 180,E1 -13854.206,E2 -13854.206} C_VEL
LIN {X 0,Y 348.201,Z 274.73,A -85,B 0,C 180,E1 -13857.687,E2 -13857.687} C_VEL
LIN {X 0,Y 348.339,Z 274.716,A -85,B 0,C 180,E1 -13860,E2 -13860} C_VEL
LIN {X 0,Y 348.201,Z 274.716,A -85,B 0,C 180,E1 -13862.314,E2 -13862.314} C_VEL
LIN {X 0,Y 348.085,Z 274.749,A -85,B 0,C 180,E1 -13866.958,E2 -13866.958} C_VEL
LIN {X 0,Y 347.922,Z 274.764,A -85,B 0,C 180,E1 -13870.475,E2 -13870.475} C_VEL
LIN {X 0,Y 347.893,Z 274.763,A -85,B 0,C 180,E1 -13874.15,E2 -13874.15} C_VEL
LIN {X 0,Y 347.885,Z 274.774,A -85,B 0,C 180,E1 -13878.29,E2 -13878.29} C_VEL
LIN {X 0,Y 347.783,Z 274.779,A -85,B 0,C 180,E1 -13881.635,E2 -13881.635} C_VEL
LIN {X 0,Y 347.807,Z 274.778,A -85,B 0,C 180,E1 -13885.109,E2 -13885.109} C_VEL
LIN {X 0,Y 347.807,Z 274.783,A -85,B 0,C 180,E1 -13887.694,E2 -13887.694} C_VEL
LIN {X 0,Y 347.76,Z 274.786,A -85,B 0,C 180,E1 -13890.347,E2 -13890.347} C_VEL
LIN {X 0,Y 347.74,Z 274.754,A -85,B 0,C 180,E1 -13894.465,E2 -13894.465} C_VEL
LIN {X 0,Y 347.774,Z 274.789,A -85,B 0,C 180,E1 -13897.99,E2 -13897.99} C_VEL
LIN {X 0,Y 347.754,Z 274.758,A -85,B 0,C 180,E1 -13901.83,E2 -13901.83} C_VEL
LIN {X 0,Y 347.764,Z 274.792,A -85,B 0,C 180,E1 -13905.017,E2 -13905.017} C_VEL
LIN {X 0,Y 347.748,Z 274.772,A -85,B 0,C 180,E1 -13908.398,E2 -13908.398} C_VEL
LIN {X 0,Y 347.772,Z 274.776,A -85,B 0,C 180,E1 -13912.012,E2 -13912.012} C_VEL
LIN {X 0,Y 347.743,Z 274.784,A -85,B 0,C 180,E1 -13915.537,E2 -13915.537} C_VEL
LIN {X 0,Y 347.753,Z 274.894,A -85,B 0,C 180,E1 -13918.083,E2 -13918.083} C_VEL
LIN {X 0,Y 350.429,Z 285.724,A -85,B 0,C 180,E1 -13921.228,E2 -13921.228} C_VEL
LIN {X 0,Y 351.149,Z 288.694,A -85,B 0,C 180,E1 -13921.951,E2 -13921.951} C_VEL
LIN {X 0,Y 359.286,Z 308.318,A -85,B 0,C 180,E1 -13923.094,E2 -13923.094} C_VEL
LIN {X 0,Y 362.232,Z 323.194,A -85,B 0,C 180,E1 -13923.654,E2 -13923.654} C_VEL
LIN {X 0,Y 360.472,Z 405.355,A -85,B 0,C 180,E1 -13925.295,E2 -13925.295} C_VEL
LIN {X 0,Y 359.807,Z 427.658,A -85,B 0,C 180,E1 -13925.784,E2 -13925.784} C_VEL
LIN {X 0,Y 359,Z 441.525,A -85,B 0,C 180,E1 -13926.301,E2 -13926.301} C_VEL
LIN {X 0,Y 357.914,Z 455.08,A -85,B 0,C 180,E1 -13927.029,E2 -13927.029} C_VEL
LIN {X 0,Y 356.633,Z 468.696,A -85,B 0,C 180,E1 -13928.012,E2 -13928.012} C_VEL
LIN {X 0,Y 355.218,Z 480.923,A -85,B 0,C 180,E1 -13929.138,E2 -13929.138} C_VEL
LIN {X 0,Y 353.566,Z 493.251,A -85,B 0,C 180,E1 -13930.553,E2 -13930.553} C_VEL
LIN {X 0,Y 352.116,Z 503.384,A -85,B 0,C 180,E1 -13931.979,E2 -13931.979} C_VEL
LIN {X 0,Y 350.507,Z 513.442,A -85,B 0,C 180,E1 -13933.698,E2 -13933.698} C_VEL
LIN {X 0,Y 349.395,Z 521.791,A -85,B 0,C 180,E1 -13935.438,E2 -13935.438} C_VEL
LIN {X 0,Y 348.405,Z 528.759,A -85,B 0,C 180,E1 -13937.18,E2 -13937.18} C_VEL
LIN {X 0,Y 347.566,Z 534.508,A -85,B 0,C 180,E1 -13938.925,E2 -13938.925} C_VEL
LIN {X 0,Y 346.959,Z 539.236,A -85,B 0,C 180,E1 -13940.674,E2 -13940.674} C_VEL
LIN {X 0,Y 346.525,Z 544.131,A -85,B 0,C 180,E1 -13943.011,E2 -13943.011} C_VEL
LIN {X 0,Y 346.257,Z 547.539,A -85,B 0,C 180,E1 -13945.343,E2 -13945.343} C_VEL
LIN {X 0,Y 346.084,Z 549.564,A -85,B 0,C 180,E1 -13947.672,E2 -13947.672} C_VEL
LIN {X 0,Y 346.075,Z 550.257,A -85,B 0,C 180,E1 -13950,E2 -13950} C_VEL
LIN {X 0,Y 346.083,Z 549.629,A -85,B 0,C 180,E1 -13952.328,E2 -13952.328} C_VEL
LIN {X 0,Y 346.258,Z 547.664,A -85,B 0,C 180,E1 -13954.657,E2 -13954.657} C_VEL
LIN {X 0,Y 346.525,Z 544.317,A -85,B 0,C 180,E1 -13956.989,E2 -13956.989} C_VEL
LIN {X 0,Y 346.946,Z 539.489,A -85,B 0,C 180,E1 -13959.326,E2 -13959.326} C_VEL
LIN {X 0,Y 347.725,Z 533.025,A -85,B 0,C 180,E1 -13961.66,E2 -13961.66} C_VEL
LIN {X 0,Y 348.859,Z 525.826,A -85,B 0,C 180,E1 -13963.692,E2 -13963.692} C_VEL
LIN {X 0,Y 350.073,Z 516.925,A -85,B 0,C 180,E1 -13965.724,E2 -13965.724} C_VEL
LIN {X 0,Y 351.46,Z 507.566,A -85,B 0,C 180,E1 -13967.454,E2 -13967.454} C_VEL
LIN {X 0,Y 352.984,Z 497.204,A -85,B 0,C 180,E1 -13969.027,E2 -13969.027} C_VEL
LIN {X 0,Y 354.624,Z 485.768,A -85,B 0,C 180,E1 -13970.444,E2 -13970.444} C_VEL
LIN {X 0,Y 356.185,Z 473.091,A -85,B 0,C 180,E1 -13971.713,E2 -13971.713} C_VEL
LIN {X 0,Y 357.436,Z 460.766,A -85,B 0,C 180,E1 -13972.697,E2 -13972.697} C_VEL
LIN {X 0,Y 358.602,Z 447.085,A -85,B 0,C 180,E1 -13973.535,E2 -13973.535} C_VEL
LIN {X 0,Y 359.526,Z 433.901,A -85,B 0,C 180,E1 -13974.115,E2 -13974.115} C_VEL
LIN {X 0,Y 359.337,Z 428.186,A -85,B 0,C 180,E1 -13974.343,E2 -13974.343} C_VEL
LIN {X 0,Y 357.091,Z 418.914,A -85,B 0,C 180,E1 -13974.771,E2 -13974.771} C_VEL
LIN {X 0,Y 354.653,Z 409.586,A -85,B 0,C 180,E1 -13975.159,E2 -13975.159} C_VEL
LIN {X 0,Y 354.164,Z 403.773,A -85,B 0,C 180,E1 -13975.32,E2 -13975.32} C_VEL
LIN {X 0,Y 355.862,Z 324.246,A -85,B 0,C 180,E1 -13976.942,E2 -13976.942} C_VEL
LIN {X 0,Y 353.099,Z 310.432,A -85,B 0,C 180,E1 -13977.48,E2 -13977.48} C_VEL
LIN {X 0,Y 344.843,Z 290.974,A -85,B 0,C 180,E1 -13978.649,E2 -13978.649} C_VEL
LIN {X 0,Y 343.763,Z 288.258,A -85,B 0,C 180,E1 -13978.879,E2 -13978.879} C_VEL
LIN {X 0,Y 341.038,Z 277.057,A -85,B 0,C 180,E1 -13982.109,E2 -13982.109} C_VEL
LIN {X 0,Y 340.702,Z 275.699,A -85,B 0,C 180,E1 -13982.63,E2 -13982.63} C_VEL
LIN {X 0,Y 340.716,Z 275.667,A -85,B 0,C 180,E1 -13985.278,E2 -13985.278} C_VEL
LIN {X 0,Y 340.708,Z 275.658,A -85,B 0,C 180,E1 -13988.385,E2 -13988.385} C_VEL
LIN {X 0,Y 340.696,Z 275.649,A -85,B 0,C 180,E1 -13992.045,E2 -13992.045} C_VEL
LIN {X 0,Y 340.682,Z 275.674,A -85,B 0,C 180,E1 -13995.461,E2 -13995.461} C_VEL
LIN {X 0,Y 340.69,Z 275.638,A -85,B 0,C 180,E1 -13998.691,E2 -13998.691} C_VEL
LIN {X 0,Y 340.731,Z 275.671,A -85,B 0,C 180,E1 -14001.772,E2 -14001.772} C_VEL
LIN {X 0,Y 340.718,Z 275.632,A -85,B 0,C 180,E1 -14005.595,E2 -14005.595} C_VEL
LIN {X 0,Y 340.699,Z 275.653,A -85,B 0,C 180,E1 -14008.955,E2 -14008.955} C_VEL
LIN {X 0,Y 340.774,Z 275.661,A -85,B 0,C 180,E1 -14012.473,E2 -14012.473} C_VEL
LIN {X 0,Y 340.75,Z 275.664,A -85,B 0,C 180,E1 -14015.638,E2 -14015.638} C_VEL
LIN {X 0,Y 340.738,Z 275.653,A -85,B 0,C 180,E1 -14019.473,E2 -14019.473} C_VEL
LIN {X 0,Y 340.851,Z 275.651,A -85,B 0,C 180,E1 -14021.984,E2 -14021.984} C_VEL
LIN {X 0,Y 340.863,Z 275.638,A -85,B 0,C 180,E1 -14025.705,E2 -14025.705} C_VEL
LIN {X 0,Y 340.864,Z 275.644,A -85,B 0,C 180,E1 -14029.306,E2 -14029.306} C_VEL
LIN {X 0,Y 341.053,Z 275.621,A -85,B 0,C 180,E1 -14032.898,E2 -14032.898} C_VEL
LIN {X 0,Y 341.163,Z 275.592,A -85,B 0,C 180,E1 -14037.639,E2 -14037.639} C_VEL
LIN {X 0,Y 341.31,Z 275.591,A -85,B 0,C 180,E1 -14040,E2 -14040} C_VEL
LIN {X 0,Y 341.162,Z 275.606,A -85,B 0,C 180,E1 -14042.361,E2 -14042.361} C_VEL
LIN {X 0,Y 341.068,Z 275.623,A -85,B 0,C 180,E1 -14047.102,E2 -14047.102} C_VEL
LIN {X 0,Y 340.863,Z 275.635,A -85,B 0,C 180,E1 -14050.694,E2 -14050.694} C_VEL
LIN {X 0,Y 340.856,Z 275.649,A -85,B 0,C 180,E1 -14054.325,E2 -14054.325} C_VEL
LIN {X 0,Y 340.83,Z 275.654,A -85,B 0,C 180,E1 -14058.467,E2 -14058.467} C_VEL
LIN {X 0,Y 340.747,Z 275.652,A -85,B 0,C 180,E1 -14061.857,E2 -14061.857} C_VEL
LIN {X 0,Y 340.766,Z 275.663,A -85,B 0,C 180,E1 -14065.665,E2 -14065.665} C_VEL
LIN {X 0,Y 340.736,Z 275.659,A -85,B 0,C 180,E1 -14068.32,E2 -14068.32} C_VEL
LIN {X 0,Y 340.699,Z 275.668,A -85,B 0,C 180,E1 -14071.045,E2 -14071.045} C_VEL
LIN {X 0,Y 340.713,Z 275.629,A -85,B 0,C 180,E1 -14075.279,E2 -14075.279} C_VEL
LIN {X 0,Y 340.705,Z 275.671,A -85,B 0,C 180,E1 -14078.387,E2 -14078.387} C_VEL
LIN {X 0,Y 340.695,Z 275.674,A -85,B 0,C 180,E1 -14082.046,E2 -14082.046} C_VEL
LIN {X 0,Y 340.732,Z 275.668,A -85,B 0,C 180,E1 -14085.471,E2 -14085.471} C_VEL
LIN {X 0,Y 340.721,Z 275.644,A -85,B 0,C 180,E1 -14088.697,E2 -14088.697} C_VEL
LIN {X 0,Y 340.736,Z 275.658,A -85,B 0,C 180,E1 -14091.774,E2 -14091.774} C_VEL
LIN {X 0,Y 340.709,Z 275.659,A -85,B 0,C 180,E1 -14095.876,E2 -14095.876} C_VEL
LIN {X 0,Y 340.757,Z 275.867,A -85,B 0,C 180,E1 -14096.259,E2 -14096.259} C_VEL
LIN {X 0,Y 343.9,Z 288.767,A -85,B 0,C 180,E1 -14099.955,E2 -14099.955} C_VEL
LIN {X 0,Y 345.145,Z 294.127,A -85,B 0,C 180,E1 -14101.336,E2 -14101.336} C_VEL
LIN {X 0,Y 351.207,Z 308.802,A -85,B 0,C 180,E1 -14102.235,E2 -14102.235} C_VEL
LIN {X 0,Y 355.751,Z 332.637,A -85,B 0,C 180,E1 -14103.148,E2 -14103.148} C_VEL
LIN {X 0,Y 353.587,Z 426.495,A -85,B 0,C 180,E1 -14105.056,E2 -14105.056} C_VEL
LIN {X 0,Y 352.826,Z 441.521,A -85,B 0,C 180,E1 -14105.509,E2 -14105.509} C_VEL
LIN {X 0,Y 351.764,Z 455.029,A -85,B 0,C 180,E1 -14106.136,E2 -14106.136} C_VEL
LIN {X 0,Y 350.492,Z 468.283,A -85,B 0,C 180,E1 -14106.983,E2 -14106.983} C_VEL
LIN {X 0,Y 349.034,Z 481.534,A -85,B 0,C 180,E1 -14108.091,E2 -14108.091} C_VEL
LIN {X 0,Y 347.337,Z 494.079,A -85,B 0,C 180,E1 -14109.418,E2 -14109.418} C_VEL
LIN {X 0,Y 345.835,Z 504.141,A -85,B 0,C 180,E1 -14110.718,E2 -14110.718} C_VEL
LIN {X 0,Y 344.12,Z 515.206,A -85,B 0,C 180,E1 -14112.468,E2 -14112.468} C_VEL
LIN {X 0,Y 342.751,Z 524.337,A -85,B 0,C 180,E1 -14114.236,E2 -14114.236} C_VEL
LIN {X 0,Y 341.517,Z 533.064,A -85,B 0,C 180,E1 -14116.311,E2 -14116.311} C_VEL
LIN {X 0,Y 340.524,Z 539.207,A -85,B 0,C 180,E1 -14118.09,E2 -14118.09} C_VEL
LIN {X 0,Y 339.733,Z 545.734,A -85,B 0,C 180,E1 -14120.474,E2 -14120.474} C_VEL
LIN {X 0,Y 339.29,Z 550.618,A -85,B 0,C 180,E1 -14122.861,E2 -14122.861} C_VEL
LIN {X 0,Y 339.064,Z 554.013,A -85,B 0,C 180,E1 -14125.244,E2 -14125.244} C_VEL
LIN {X 0,Y 338.961,Z 556.02,A -85,B 0,C 180,E1 -14127.624,E2 -14127.624} C_VEL
LIN {X 0,Y 338.977,Z 556.683,A -85,B 0,C 180,E1 -14130,E2 -14130} C_VEL
LIN {X 0,Y 338.961,Z 556.012,A -85,B 0,C 180,E1 -14132.377,E2 -14132.377} C_VEL
LIN {X 0,Y 339.065,Z 553.999,A -85,B 0,C 180,E1 -14134.756,E2 -14134.756} C_VEL
LIN {X 0,Y 339.29,Z 550.594,A -85,B 0,C 180,E1 -14137.139,E2 -14137.139} C_VEL
LIN {X 0,Y 339.737,Z 545.696,A -85,B 0,C 180,E1 -14139.526,E2 -14139.526} C_VEL
LIN {X 0,Y 340.524,Z 539.159,A -85,B 0,C 180,E1 -14141.911,E2 -14141.911} C_VEL
LIN {X 0,Y 341.509,Z 533.006,A -85,B 0,C 180,E1 -14143.689,E2 -14143.689} C_VEL
LIN {X 0,Y 342.689,Z 524.264,A -85,B 0,C 180,E1 -14145.767,E2 -14145.767} C_VEL
LIN {X 0,Y 344.101,Z 515.119,A -85,B 0,C 180,E1 -14147.533,E2 -14147.533} C_VEL
LIN {X 0,Y 345.784,Z 504.026,A -85,B 0,C 180,E1 -14149.285,E2 -14149.285} C_VEL
LIN {X 0,Y 347.538,Z 492.701,A -85,B 0,C 180,E1 -14150.725,E2 -14150.725} C_VEL
LIN {X 0,Y 349.034,Z 481.369,A -85,B 0,C 180,E1 -14151.908,E2 -14151.908} C_VEL
LIN {X 0,Y 350.346,Z 470.028,A -85,B 0,C 180,E1 -14152.871,E2 -14152.871} C_VEL
LIN {X 0,Y 351.587,Z 457.311,A -85,B 0,C 180,E1 -14153.721,E2 -14153.721} C_VEL
LIN {X 0,Y 352.688,Z 442.924,A -85,B 0,C 180,E1 -14154.423,E2 -14154.423} C_VEL
LIN {X 0,Y 353.474,Z 428.816,A -85,B 0,C 180,E1 -14154.875,E2 -14154.875} C_VEL
LIN {X 0,Y 355.775,Z 333.428,A -85,B 0,C 180,E1 -14156.814,E2 -14156.814} C_VEL
LIN {X 0,Y 351.163,Z 308.689,A -85,B 0,C 180,E1 -14157.752,E2 -14157.752} C_VEL
LIN {X 0,Y 345.116,Z 294.004,A -85,B 0,C 180,E1 -14158.657,E2 -14158.657} C_VEL
LIN {X 0,Y 342.291,Z 281.976,A -85,B 0,C 180,E1 -14161.917,E2 -14161.917} C_VEL
LIN {X 0,Y 340.729,Z 275.813,A -85,B 0,C 180,E1 -14163.753,E2 -14163.753} C_VEL
LIN {X 0,Y 340.702,Z 275.655,A -85,B 0,C 180,E1 -14166.741,E2 -14166.741} C_VEL
LIN {X 0,Y 340.685,Z 275.66,A -85,B 0,C 180,E1 -14170.246,E2 -14170.246} C_VEL
LIN {X 0,Y 340.649,Z 275.675,A -85,B 0,C 180,E1 -14173.773,E2 -14173.773} C_VEL
LIN {X 0,Y 340.695,Z 275.673,A -85,B 0,C 180,E1 -14177.954,E2 -14177.954} C_VEL
LIN {X 0,Y 340.729,Z 275.669,A -85,B 0,C 180,E1 -14181.772,E2 -14181.772} C_VEL
LIN {X 0,Y 340.718,Z 275.623,A -85,B 0,C 180,E1 -14185.595,E2 -14185.595} C_VEL
LIN {X 0,Y 340.699,Z 275.668,A -85,B 0,C 180,E1 -14188.956,E2 -14188.956} C_VEL
LIN {X 0,Y 340.774,Z 275.649,A -85,B 0,C 180,E1 -14192.473,E2 -14192.473} C_VEL
LIN {X 0,Y 340.766,Z 275.664,A -85,B 0,C 180,E1 -14195.639,E2 -14195.639} C_VEL
LIN {X 0,Y 340.747,Z 275.66,A -85,B 0,C 180,E1 -14199.474,E2 -14199.474} C_VEL
LIN {X 0,Y 340.852,Z 275.645,A -85,B 0,C 180,E1 -14201.984,E2 -14201.984} C_VEL
LIN {X 0,Y 340.863,Z 275.649,A -85,B 0,C 180,E1 -14205.705,E2 -14205.705} C_VEL
LIN {X 0,Y 340.864,Z 275.635,A -85,B 0,C 180,E1 -14209.306,E2 -14209.306} C_VEL
LIN {X 0,Y 341.068,Z 275.623,A -85,B 0,C 180,E1 -14212.898,E2 -14212.898} C_VEL
LIN {X 0,Y 341.163,Z 275.606,A -85,B 0,C 180,E1 -14217.639,E2 -14217.639} C_VEL
LIN {X 0,Y 341.289,Z 275.594,A -85,B 0,C 180,E1 -14220,E2 -14220} C_VEL
LIN {X 0,Y 341.163,Z 275.592,A -85,B 0,C 180,E1 -14222.361,E2 -14222.361} C_VEL
LIN {X 0,Y 341.053,Z 275.622,A -85,B 0,C 180,E1 -14227.102,E2 -14227.102} C_VEL
LIN {X 0,Y 340.864,Z 275.644,A -85,B 0,C 180,E1 -14230.694,E2 -14230.694} C_VEL
LIN {X 0,Y 340.857,Z 275.639,A -85,B 0,C 180,E1 -14234.325,E2 -14234.325} C_VEL
LIN {X 0,Y 340.831,Z 275.654,A -85,B 0,C 180,E1 -14238.467,E2 -14238.467} C_VEL
LIN {X 0,Y 340.749,Z 275.657,A -85,B 0,C 180,E1 -14241.857,E2 -14241.857} C_VEL
LIN {X 0,Y 340.767,Z 275.65,A -85,B 0,C 180,E1 -14245.665,E2 -14245.665} C_VEL
LIN {X 0,Y 340.738,Z 275.664,A -85,B 0,C 180,E1 -14248.32,E2 -14248.32} C_VEL
LIN {X 0,Y 340.7,Z 275.653,A -85,B 0,C 180,E1 -14251.045,E2 -14251.045} C_VEL
LIN {X 0,Y 340.715,Z 275.641,A -85,B 0,C 180,E1 -14255.279,E2 -14255.279} C_VEL
LIN {X 0,Y 340.711,Z 275.671,A -85,B 0,C 180,E1 -14258.388,E2 -14258.388} C_VEL
LIN {X 0,Y 340.701,Z 275.637,A -85,B 0,C 180,E1 -14262.047,E2 -14262.047} C_VEL
LIN {X 0,Y 340.681,Z 275.671,A -85,B 0,C 180,E1 -14265.462,E2 -14265.462} C_VEL
LIN {X 0,Y 340.684,Z 275.655,A -85,B 0,C 180,E1 -14268.691,E2 -14268.691} C_VEL
LIN {X 0,Y 340.732,Z 275.654,A -85,B 0,C 180,E1 -14271.773,E2 -14271.773} C_VEL
LIN {X 0,Y 340.722,Z 275.658,A -85,B 0,C 180,E1 -14275.596,E2 -14275.596} C_VEL
LIN {X 0,Y 340.725,Z 275.781,A -85,B 0,C 180,E1 -14277.569,E2 -14277.569} C_VEL
LIN {X 0,Y 343.157,Z 285.797,A -85,B 0,C 180,E1 -14280.559,E2 -14280.559} C_VEL
LIN {X 0,Y 343.915,Z 288.732,A -85,B 0,C 180,E1 -14281.303,E2 -14281.303} C_VEL
LIN {X 0,Y 351.798,Z 307.203,A -85,B 0,C 180,E1 -14282.446,E2 -14282.446} C_VEL
LIN {X 0,Y 353.418,Z 311.725,A -85,B 0,C 180,E1 -14282.685,E2 -14282.685} C_VEL
LIN {X 0,Y 355.954,Z 324.915,A -85,B 0,C 180,E1 -14283.189,E2 -14283.189} C_VEL
LIN {X 0,Y 353.922,Z 409.023,A -85,B 0,C 180,E1 -14284.884,E2 -14284.884} C_VEL
LIN {X 0,Y 353.283,Z 428.879,A -85,B 0,C 180,E1 -14285.346,E2 -14285.346} C_VEL
LIN {X 0,Y 352.396,Z 443.125,A -85,B 0,C 180,E1 -14285.908,E2 -14285.908} C_VEL
LIN {X 0,Y 351.26,Z 456.629,A -85,B 0,C 180,E1 -14286.67,E2 -14286.67} C_VEL
LIN {X 0,Y 349.96,Z 469.687,A -85,B 0,C 180,E1 -14287.651,E2 -14287.651} C_VEL
LIN {X 0,Y 348.392,Z 482.359,A -85,B 0,C 180,E1 -14288.864,E2 -14288.864} C_VEL
LIN {X 0,Y 346.673,Z 494.389,A -85,B 0,C 180,E1 -14290.304,E2 -14290.304} C_VEL
LIN {X 0,Y 345.059,Z 505.233,A -85,B 0,C 180,E1 -14291.905,E2 -14291.905} C_VEL
LIN {X 0,Y 343.443,Z 514.996,A -85,B 0,C 180,E1 -14293.659,E2 -14293.659} C_VEL
LIN {X 0,Y 342.343,Z 523.182,A -85,B 0,C 180,E1 -14295.458,E2 -14295.458} C_VEL
LIN {X 0,Y 341.079,Z 530.84,A -85,B 0,C 180,E1 -14297.505,E2 -14297.505} C_VEL
LIN {X 0,Y 340.34,Z 536.254,A -85,B 0,C 180,E1 -14299.29,E2 -14299.29} C_VEL
LIN {X 0,Y 339.61,Z 541.946,A -85,B 0,C 180,E1 -14301.671,E2 -14301.671} C_VEL
LIN {X 0,Y 339.279,Z 546.082,A -85,B 0,C 180,E1 -14304.055,E2 -14304.055} C_VEL
LIN {X 0,Y 339.088,Z 548.787,A -85,B 0,C 180,E1 -14306.435,E2 -14306.435} C_VEL
LIN {X 0,Y 338.966,Z 550.142,A -85,B 0,C 180,E1 -14308.812,E2 -14308.812} C_VEL
LIN {X 0,Y 338.966,Z 550.175,A -85,B 0,C 180,E1 -14311.188,E2 -14311.188} C_VEL
LIN {X 0,Y 339.088,Z 548.882,A -85,B 0,C 180,E1 -14313.565,E2 -14313.565} C_VEL
LIN {X 0,Y 339.278,Z 546.234,A -85,B 0,C 180,E1 -14315.945,E2 -14315.945} C_VEL
LIN {X 0,Y 339.608,Z 542.163,A -85,B 0,C 180,E1 -14318.329,E2 -14318.329} C_VEL
LIN {X 0,Y 340.314,Z 536.538,A -85,B 0,C 180,E1 -14320.711,E2 -14320.711} C_VEL
LIN {X 0,Y 341.24,Z 530.187,A -85,B 0,C 180,E1 -14322.791,E2 -14322.791} C_VEL
LIN {X 0,Y 342.361,Z 522.476,A -85,B 0,C 180,E1 -14324.822,E2 -14324.822} C_VEL
LIN {X 0,Y 343.656,Z 514.028,A -85,B 0,C 180,E1 -14326.637,E2 -14326.637} C_VEL
LIN {X 0,Y 345.226,Z 504.073,A -85,B 0,C 180,E1 -14328.393,E2 -14328.393} C_VEL
LIN {X 0,Y 346.922,Z 492.991,A -85,B 0,C 180,E1 -14329.989,E2 -14329.989} C_VEL
LIN {X 0,Y 348.659,Z 480.614,A -85,B 0,C 180,E1 -14331.422,E2 -14331.422} C_VEL
LIN {X 0,Y 350.219,Z 467.686,A -85,B 0,C 180,E1 -14332.615,E2 -14332.615} C_VEL
LIN {X 0,Y 351.514,Z 454.472,A -85,B 0,C 180,E1 -14333.569,E2 -14333.569} C_VEL
LIN {X 0,Y 352.604,Z 440.668,A -85,B 0,C 180,E1 -14334.312,E2 -14334.312} C_VEL
LIN {X 0,Y 353.45,Z 426.325,A -85,B 0,C 180,E1 -14334.837,E2 -14334.837} C_VEL
LIN {X 0,Y 354.164,Z 403.773,A -85,B 0,C 180,E1 -14335.32,E2 -14335.32} C_VEL
LIN {X 0,Y 353.685,Z 397.962,A -85,B 0,C 180,E1 -14335.485,E2 -14335.485} C_VEL
LIN {X 0,Y 348.9,Z 379.302,A -85,B 0,C 180,E1 -14336.28,E2 -14336.28} C_VEL
LIN {X 0,Y 348.51,Z 373.49,A -85,B 0,C 180,E1 -14336.443,E2 -14336.443} C_VEL
LIN {X 0,Y 349.492,Z 324.817,A -85,B 0,C 180,E1 -14337.462,E2 -14337.462} C_VEL
LIN {X 0,Y 346.942,Z 312.683,A -85,B 0,C 180,E1 -14337.96,E2 -14337.96} C_VEL
LIN {X 0,Y 338.755,Z 293.434,A -85,B 0,C 180,E1 -14339.155,E2 -14339.155} C_VEL
LIN {X 0,Y 336.554,Z 288.405,A -85,B 0,C 180,E1 -14339.546,E2 -14339.546} C_VEL
LIN {X 0,Y 333.954,Z 277.859,A -85,B 0,C 180,E1 -14342.67,E2 -14342.67} C_VEL
LIN {X 0,Y 333.682,Z 276.566,A -85,B 0,C 180,E1 -14343.202,E2 -14343.202} C_VEL
LIN {X 0,Y 333.663,Z 276.54,A -85,B 0,C 180,E1 -14346.831,E2 -14346.831} C_VEL
LIN {X 0,Y 333.644,Z 276.544,A -85,B 0,C 180,E1 -14350.767,E2 -14350.767} C_VEL
LIN {X 0,Y 333.622,Z 276.548,A -85,B 0,C 180,E1 -14354.255,E2 -14354.255} C_VEL
LIN {X 0,Y 333.642,Z 276.521,A -85,B 0,C 180,E1 -14357.618,E2 -14357.618} C_VEL
LIN {X 0,Y 333.651,Z 276.545,A -85,B 0,C 180,E1 -14361.201,E2 -14361.201} C_VEL
LIN {X 0,Y 333.672,Z 276.541,A -85,B 0,C 180,E1 -14363.86,E2 -14363.86} C_VEL
LIN {X 0,Y 333.638,Z 276.508,A -85,B 0,C 180,E1 -14367.412,E2 -14367.412} C_VEL
LIN {X 0,Y 333.706,Z 276.545,A -85,B 0,C 180,E1 -14371.027,E2 -14371.027} C_VEL
LIN {X 0,Y 333.73,Z 276.525,A -85,B 0,C 180,E1 -14373.753,E2 -14373.753} C_VEL
LIN {X 0,Y 333.714,Z 276.536,A -85,B 0,C 180,E1 -14377.913,E2 -14377.913} C_VEL
LIN {X 0,Y 333.787,Z 276.531,A -85,B 0,C 180,E1 -14381.589,E2 -14381.589} C_VEL
LIN {X 0,Y 333.802,Z 276.516,A -85,B 0,C 180,E1 -14385.576,E2 -14385.576} C_VEL
LIN {X 0,Y 333.827,Z 276.522,A -85,B 0,C 180,E1 -14389.078,E2 -14389.078} C_VEL
LIN {X 0,Y 334,Z 276.497,A -85,B 0,C 180,E1 -14392.747,E2 -14392.747} C_VEL
LIN {X 0,Y 333.805,Z 276.527,A -85,B 0,C 180,E1 -14395.169,E2 -14395.169} C_VEL
LIN {X 0,Y 334.1,Z 276.472,A -85,B 0,C 180,E1 -14397.589,E2 -14397.589} C_VEL
LIN {X 0,Y 334.26,Z 276.469,A -85,B 0,C 180,E1 -14400,E2 -14400} C_VEL
LIN {X 0,Y 334.099,Z 276.485,A -85,B 0,C 180,E1 -14402.411,E2 -14402.411} C_VEL
LIN {X 0,Y 334.018,Z 276.501,A -85,B 0,C 180,E1 -14407.253,E2 -14407.253} C_VEL
LIN {X 0,Y 333.826,Z 276.513,A -85,B 0,C 180,E1 -14410.922,E2 -14410.922} C_VEL
LIN {X 0,Y 333.801,Z 276.525,A -85,B 0,C 180,E1 -14414.634,E2 -14414.634} C_VEL
LIN {X 0,Y 333.789,Z 276.532,A -85,B 0,C 180,E1 -14418.655,E2 -14418.655} C_VEL
LIN {X 0,Y 333.686,Z 276.531,A -85,B 0,C 180,E1 -14422.279,E2 -14422.279} C_VEL
LIN {X 0,Y 333.73,Z 276.531,A -85,B 0,C 180,E1 -14426.247,E2 -14426.247} C_VEL
LIN {X 0,Y 333.706,Z 276.539,A -85,B 0,C 180,E1 -14428.973,E2 -14428.973} C_VEL
LIN {X 0,Y 333.638,Z 276.525,A -85,B 0,C 180,E1 -14432.588,E2 -14432.588} C_VEL
LIN {X 0,Y 333.671,Z 276.518,A -85,B 0,C 180,E1 -14436.14,E2 -14436.14} C_VEL
LIN {X 0,Y 333.642,Z 276.55,A -85,B 0,C 180,E1 -14439.193,E2 -14439.193} C_VEL
LIN {X 0,Y 333.63,Z 276.551,A -85,B 0,C 180,E1 -14442.501,E2 -14442.501} C_VEL
LIN {X 0,Y 333.669,Z 276.546,A -85,B 0,C 180,E1 -14445.968,E2 -14445.968} C_VEL
LIN {X 0,Y 333.698,Z 276.523,A -85,B 0,C 180,E1 -14449.305,E2 -14449.305} C_VEL
LIN {X 0,Y 333.663,Z 276.531,A -85,B 0,C 180,E1 -14453.168,E2 -14453.168} C_VEL
LIN {X 0,Y 333.72,Z 276.767,A -85,B 0,C 180,E1 -14455.714,E2 -14455.714} C_VEL
LIN {X 0,Y 336.382,Z 287.642,A -85,B 0,C 180,E1 -14458.938,E2 -14458.938} C_VEL
LIN {X 0,Y 337.857,Z 293.973,A -85,B 0,C 180,E1 -14460.651,E2 -14460.651} C_VEL
LIN {X 0,Y 344.54,Z 309.588,A -85,B 0,C 180,E1 -14461.669,E2 -14461.669} C_VEL
LIN {X 0,Y 345.707,Z 313.792,A -85,B 0,C 180,E1 -14461.87,E2 -14461.87} C_VEL
LIN {X 0,Y 349.461,Z 334.152,A -85,B 0,C 180,E1 -14462.66,E2 -14462.66} C_VEL
LIN {X 0,Y 347.049,Z 429.456,A -85,B 0,C 180,E1 -14464.633,E2 -14464.633} C_VEL
LIN {X 0,Y 346.183,Z 444.197,A -85,B 0,C 180,E1 -14465.127,E2 -14465.127} C_VEL
LIN {X 0,Y 344.948,Z 458.672,A -85,B 0,C 180,E1 -14465.874,E2 -14465.874} C_VEL
LIN {X 0,Y 343.573,Z 471.946,A -85,B 0,C 180,E1 -14466.811,E2 -14466.811} C_VEL
LIN {X 0,Y 342.155,Z 483.686,A -85,B 0,C 180,E1 -14467.868,E2 -14467.868} C_VEL
LIN {X 0,Y 340.32,Z 496.365,A -85,B 0,C 180,E1 -14469.29,E2 -14469.29} C_VEL
LIN {X 0,Y 338.803,Z 506.044,A -85,B 0,C 180,E1 -14470.617,E2 -14470.617} C_VEL
LIN {X 0,Y 337.053,Z 516.771,A -85,B 0,C 180,E1 -14472.402,E2 -14472.402} C_VEL
LIN {X 0,Y 335.635,Z 525.628,A -85,B 0,C 180,E1 -14474.204,E2 -14474.204} C_VEL
LIN {X 0,Y 334.425,Z 534.116,A -85,B 0,C 180,E1 -14476.325,E2 -14476.325} C_VEL
LIN {X 0,Y 333.281,Z 540.954,A -85,B 0,C 180,E1 -14478.444,E2 -14478.444} C_VEL
LIN {X 0,Y 332.709,Z 545.668,A -85,B 0,C 180,E1 -14480.271,E2 -14480.271} C_VEL
LIN {X 0,Y 332.238,Z 550.552,A -85,B 0,C 180,E1 -14482.709,E2 -14482.709} C_VEL
LIN {X 0,Y 331.975,Z 553.947,A -85,B 0,C 180,E1 -14485.143,E2 -14485.143} C_VEL
LIN {X 0,Y 331.881,Z 555.954,A -85,B 0,C 180,E1 -14487.573,E2 -14487.573} C_VEL
LIN {X 0,Y 331.883,Z 556.616,A -85,B 0,C 180,E1 -14490,E2 -14490} C_VEL
LIN {X 0,Y 331.881,Z 555.946,A -85,B 0,C 180,E1 -14492.427,E2 -14492.427} C_VEL
LIN {X 0,Y 331.976,Z 553.932,A -85,B 0,C 180,E1 -14494.858,E2 -14494.858} C_VEL
LIN {X 0,Y 332.238,Z 550.527,A -85,B 0,C 180,E1 -14497.292,E2 -14497.292} C_VEL
LIN {X 0,Y 332.713,Z 545.628,A -85,B 0,C 180,E1 -14499.729,E2 -14499.729} C_VEL
LIN {X 0,Y 333.561,Z 539.091,A -85,B 0,C 180,E1 -14502.163,E2 -14502.163} C_VEL
LIN {X 0,Y 334.537,Z 532.937,A -85,B 0,C 180,E1 -14503.98,E2 -14503.98} C_VEL
LIN {X 0,Y 335.6,Z 525.551,A -85,B 0,C 180,E1 -14505.797,E2 -14505.797} C_VEL
LIN {X 0,Y 337.04,Z 516.679,A -85,B 0,C 180,E1 -14507.599,E2 -14507.599} C_VEL
LIN {X 0,Y 338.761,Z 505.931,A -85,B 0,C 180,E1 -14509.386,E2 -14509.386} C_VEL
LIN {X 0,Y 340.509,Z 495.055,A -85,B 0,C 180,E1 -14510.856,E2 -14510.856} C_VEL
LIN {X 0,Y 342.133,Z 483.529,A -85,B 0,C 180,E1 -14512.133,E2 -14512.133} C_VEL
LIN {X 0,Y 343.586,Z 471.737,A -85,B 0,C 180,E1 -14513.188,E2 -14513.188} C_VEL
LIN {X 0,Y 344.979,Z 458.393,A -85,B 0,C 180,E1 -14514.124,E2 -14514.124} C_VEL
LIN {X 0,Y 346.123,Z 444.617,A -85,B 0,C 180,E1 -14514.838,E2 -14514.838} C_VEL
LIN {X 0,Y 347.012,Z 430.237,A -85,B 0,C 180,E1 -14515.33,E2 -14515.33} C_VEL
LIN {X 0,Y 349.431,Z 334.223,A -85,B 0,C 180,E1 -14517.321,E2 -14517.321} C_VEL
LIN {X 0,Y 345.159,Z 311.347,A -85,B 0,C 180,E1 -14518.214,E2 -14518.214} C_VEL
LIN {X 0,Y 338.763,Z 296.22,A -85,B 0,C 180,E1 -14519.152,E2 -14519.152} C_VEL
LIN {X 0,Y 337.832,Z 293.871,A -85,B 0,C 180,E1 -14519.341,E2 -14519.341} C_VEL
LIN {X 0,Y 335.072,Z 282.139,A -85,B 0,C 180,E1 -14522.626,E2 -14522.626} C_VEL
LIN {X 0,Y 333.685,Z 276.635,A -85,B 0,C 180,E1 -14524.336,E2 -14524.336} C_VEL
LIN {X 0,Y 333.65,Z 276.534,A -85,B 0,C 180,E1 -14527.651,E2 -14527.651} C_VEL
LIN {X 0,Y 333.644,Z 276.529,A -85,B 0,C 180,E1 -14530.767,E2 -14530.767} C_VEL
LIN {X 0,Y 333.591,Z 276.559,A -85,B 0,C 180,E1 -14534.25,E2 -14534.25} C_VEL
LIN {X 0,Y 333.638,Z 276.551,A -85,B 0,C 180,E1 -14537.618,E2 -14537.618} C_VEL
LIN {X 0,Y 333.649,Z 276.549,A -85,B 0,C 180,E1 -14541.201,E2 -14541.201} C_VEL
LIN {X 0,Y 333.672,Z 276.516,A -85,B 0,C 180,E1 -14543.861,E2 -14543.861} C_VEL
LIN {X 0,Y 333.639,Z 276.526,A -85,B 0,C 180,E1 -14547.413,E2 -14547.413} C_VEL
LIN {X 0,Y 333.706,Z 276.539,A -85,B 0,C 180,E1 -14551.028,E2 -14551.028} C_VEL
LIN {X 0,Y 333.73,Z 276.532,A -85,B 0,C 180,E1 -14553.753,E2 -14553.753} C_VEL
LIN {X 0,Y 333.714,Z 276.527,A -85,B 0,C 180,E1 -14557.914,E2 -14557.914} C_VEL
LIN {X 0,Y 333.788,Z 276.53,A -85,B 0,C 180,E1 -14561.589,E2 -14561.589} C_VEL
LIN {X 0,Y 333.802,Z 276.527,A -85,B 0,C 180,E1 -14565.577,E2 -14565.577} C_VEL
LIN {X 0,Y 333.827,Z 276.512,A -85,B 0,C 180,E1 -14569.078,E2 -14569.078} C_VEL
LIN {X 0,Y 334.018,Z 276.501,A -85,B 0,C 180,E1 -14572.747,E2 -14572.747} C_VEL
LIN {X 0,Y 333.804,Z 276.515,A -85,B 0,C 180,E1 -14575.169,E2 -14575.169} C_VEL
LIN {X 0,Y 334.1,Z 276.484,A -85,B 0,C 180,E1 -14577.589,E2 -14577.589} C_VEL
LIN {X 0,Y 334.24,Z 276.472,A -85,B 0,C 180,E1 -14580,E2 -14580} C_VEL
LIN {X 0,Y 334.101,Z 276.471,A -85,B 0,C 180,E1 -14582.411,E2 -14582.411} C_VEL
LIN {X 0,Y 333.986,Z 276.5,A -85,B 0,C 180,E1 -14586.649,E2 -14586.649} C_VEL
LIN {X 0,Y 333.844,Z 276.511,A -85,B 0,C 180,E1 -14589.696,E2 -14589.696} C_VEL
LIN {X 0,Y 333.79,Z 276.524,A -85,B 0,C 180,E1 -14593.392,E2 -14593.392} C_VEL
LIN {X 0,Y 333.741,Z 276.535,A -85,B 0,C 180,E1 -14597.147,E2 -14597.147} C_VEL
LIN {X 0,Y 333.73,Z 276.53,A -85,B 0,C 180,E1 -14599.691,E2 -14599.691} C_VEL
LIN {X 0,Y 333.687,Z 276.538,A -85,B 0,C 180,E1 -14602.279,E2 -14602.279} C_VEL
LIN {X 0,Y 333.731,Z 276.525,A -85,B 0,C 180,E1 -14606.247,E2 -14606.247} C_VEL
LIN {X 0,Y 333.707,Z 276.544,A -85,B 0,C 180,E1 -14608.973,E2 -14608.973} C_VEL
LIN {X 0,Y 333.639,Z 276.507,A -85,B 0,C 180,E1 -14612.588,E2 -14612.588} C_VEL
LIN {X 0,Y 333.674,Z 276.536,A -85,B 0,C 180,E1 -14616.139,E2 -14616.139} C_VEL
LIN {X 0,Y 333.665,Z 276.538,A -85,B 0,C 180,E1 -14619.19,E2 -14619.19} C_VEL
LIN {X 0,Y 333.633,Z 276.52,A -85,B 0,C 180,E1 -14622.501,E2 -14622.501} C_VEL
LIN {X 0,Y 333.62,Z 276.547,A -85,B 0,C 180,E1 -14625.96,E2 -14625.96} C_VEL
LIN {X 0,Y 333.646,Z 276.542,A -85,B 0,C 180,E1 -14629.316,E2 -14629.316} C_VEL
LIN {X 0,Y 333.664,Z 276.536,A -85,B 0,C 180,E1 -14633.168,E2 -14633.168} C_VEL
LIN {X 0,Y 333.665,Z 276.565,A -85,B 0,C 180,E1 -14636.886,E2 -14636.886} C_VEL
LIN {X 0,Y 333.709,Z 276.745,A -85,B 0,C 180,E1 -14637.072,E2 -14637.072} C_VEL
LIN {X 0,Y 336.358,Z 287.642,A -85,B 0,C 180,E1 -14640.376,E2 -14640.376} C_VEL
LIN {X 0,Y 336.694,Z 288.909,A -85,B 0,C 180,E1 -14640.636,E2 -14640.636} C_VEL
LIN {X 0,Y 342.917,Z 302.867,A -85,B 0,C 180,E1 -14641.565,E2 -14641.565} C_VEL
LIN {X 0,Y 347.352,Z 314.109,A -85,B 0,C 180,E1 -14642.22,E2 -14642.22} C_VEL
LIN {X 0,Y 349.576,Z 326.252,A -85,B 0,C 180,E1 -14642.688,E2 -14642.688} C_VEL
LIN {X 0,Y 347.585,Z 407.326,A -85,B 0,C 180,E1 -14644.354,E2 -14644.354} C_VEL
LIN {X 0,Y 346.949,Z 427.823,A -85,B 0,C 180,E1 -14644.825,E2 -14644.825} C_VEL
LIN {X 0,Y 346.058,Z 441.679,A -85,B 0,C 180,E1 -14645.357,E2 -14645.357} C_VEL
LIN {X 0,Y 344.863,Z 455.462,A -85,B 0,C 180,E1 -14646.123,E2 -14646.123} C_VEL
LIN {X 0,Y 343.481,Z 468.842,A -85,B 0,C 180,E1 -14647.123,E2 -14647.123} C_VEL
LIN {X 0,Y 341.988,Z 481.066,A -85,B 0,C 180,E1 -14648.29,E2 -14648.29} C_VEL
LIN {X 0,Y 340.341,Z 492.265,A -85,B 0,C 180,E1 -14649.607,E2 -14649.607} C_VEL
LIN {X 0,Y 338.586,Z 503.524,A -85,B 0,C 180,E1 -14651.233,E2 -14651.233} C_VEL
LIN {X 0,Y 336.858,Z 513.581,A -85,B 0,C 180,E1 -14653.017,E2 -14653.017} C_VEL
LIN {X 0,Y 335.464,Z 522.603,A -85,B 0,C 180,E1 -14654.989,E2 -14654.989} C_VEL
LIN {X 0,Y 334.34,Z 529.904,A -85,B 0,C 180,E1 -14656.94,E2 -14656.94} C_VEL
LIN {X 0,Y 333.344,Z 536.322,A -85,B 0,C 180,E1 -14659.062,E2 -14659.062} C_VEL
LIN {X 0,Y 332.573,Z 542.014,A -85,B 0,C 180,E1 -14661.493,E2 -14661.493} C_VEL
LIN {X 0,Y 332.221,Z 546.149,A -85,B 0,C 180,E1 -14663.928,E2 -14663.928} C_VEL
LIN {X 0,Y 332.018,Z 548.854,A -85,B 0,C 180,E1 -14666.359,E2 -14666.359} C_VEL
LIN {X 0,Y 331.875,Z 550.209,A -85,B 0,C 180,E1 -14668.787,E2 -14668.787} C_VEL
LIN {X 0,Y 331.875,Z 550.242,A -85,B 0,C 180,E1 -14671.213,E2 -14671.213} C_VEL
LIN {X 0,Y 332.018,Z 548.948,A -85,B 0,C 180,E1 -14673.641,E2 -14673.641} C_VEL
LIN {X 0,Y 332.219,Z 546.21,A -85,B 0,C 180,E1 -14676.133,E2 -14676.133} C_VEL
LIN {X 0,Y 332.57,Z 542.229,A -85,B 0,C 180,E1 -14678.507,E2 -14678.507} C_VEL
LIN {X 0,Y 333.321,Z 536.604,A -85,B 0,C 180,E1 -14680.939,E2 -14680.939} C_VEL
LIN {X 0,Y 334.301,Z 530.252,A -85,B 0,C 180,E1 -14683.061,E2 -14683.061} C_VEL
LIN {X 0,Y 335.384,Z 523.046,A -85,B 0,C 180,E1 -14685.01,E2 -14685.01} C_VEL
LIN {X 0,Y 336.814,Z 514.093,A -85,B 0,C 180,E1 -14686.985,E2 -14686.985} C_VEL
LIN {X 0,Y 338.45,Z 504.137,A -85,B 0,C 180,E1 -14688.775,E2 -14688.775} C_VEL
LIN {X 0,Y 340.227,Z 493.054,A -85,B 0,C 180,E1 -14690.4,E2 -14690.4} C_VEL
LIN {X 0,Y 342.038,Z 480.758,A -85,B 0,C 180,E1 -14691.849,E2 -14691.849} C_VEL
LIN {X 0,Y 343.571,Z 468.619,A -85,B 0,C 180,E1 -14692.999,E2 -14692.999} C_VEL
LIN {X 0,Y 344.897,Z 455.772,A -85,B 0,C 180,E1 -14693.962,E2 -14693.962} C_VEL
LIN {X 0,Y 346.099,Z 441.485,A -85,B 0,C 180,E1 -14694.759,E2 -14694.759} C_VEL
LIN {X 0,Y 346.968,Z 427.516,A -85,B 0,C 180,E1 -14695.293,E2 -14695.293} C_VEL
LIN {X 0,Y 347.794,Z 403.255,A -85,B 0,C 180,E1 -14695.83,E2 -14695.83} C_VEL
LIN {X 0,Y 348.51,Z 373.49,A -85,B 0,C 180,E1 -14696.443,E2 -14696.443} C_VEL
LIN {X 0,Y 348.11,Z 367.681,A -85,B 0,C 180,E1 -14696.607,E2 -14696.607} C_VEL
LIN {X 0,Y 343.337,Z 349.054,A -85,B 0,C 180,E1 -14697.437,E2 -14697.437} C_VEL
LIN {X 0,Y 342.9,Z 343.245,A -85,B 0,C 180,E1 -14697.609,E2 -14697.609} C_VEL
LIN {X 0,Y 343.172,Z 326.021,A -85,B 0,C 180,E1 -14697.985,E2 -14697.985} C_VEL
LIN {X 0,Y 340.967,Z 315.263,A -85,B 0,C 180,E1 -14698.434,E2 -14698.434} C_VEL
LIN {X 0,Y 332.342,Z 295.119,A -85,B 0,C 180,E1 -14699.734,E2 -14699.734} C_VEL
LIN {X 0,Y 329.422,Z 288.647,A -85,B 0,C 180,E1 -14700.228,E2 -14700.228} C_VEL
LIN {X 0,Y 327.062,Z 279.257,A -85,B 0,C 180,E1 -14703.066,E2 -14703.066} C_VEL
LIN {X 0,Y 326.618,Z 277.467,A -85,B 0,C 180,E1 -14703.728,E2 -14703.728} C_VEL
LIN {X 0,Y 326.626,Z 277.412,A -85,B 0,C 180,E1 -14707.238,E2 -14707.238} C_VEL
LIN {X 0,Y 326.575,Z 277.417,A -85,B 0,C 180,E1 -14711.13,E2 -14711.13} C_VEL
LIN {X 0,Y 326.554,Z 277.431,A -85,B 0,C 180,E1 -14714.747,E2 -14714.747} C_VEL
LIN {X 0,Y 326.576,Z 277.395,A -85,B 0,C 180,E1 -14718.154,E2 -14718.154} C_VEL
LIN {X 0,Y 326.622,Z 277.422,A -85,B 0,C 180,E1 -14721.391,E2 -14721.391} C_VEL
LIN {X 0,Y 326.615,Z 277.399,A -85,B 0,C 180,E1 -14724.851,E2 -14724.851} C_VEL
LIN {X 0,Y 326.603,Z 277.384,A -85,B 0,C 180,E1 -14727.455,E2 -14727.455} C_VEL
LIN {X 0,Y 326.656,Z 277.418,A -85,B 0,C 180,E1 -14730.34,E2 -14730.34} C_VEL
LIN {X 0,Y 326.684,Z 277.404,A -85,B 0,C 180,E1 -14734.516,E2 -14734.516} C_VEL
LIN {X 0,Y 326.639,Z 277.411,A -85,B 0,C 180,E1 -14738.545,E2 -14738.545} C_VEL
LIN {X 0,Y 326.738,Z 277.409,A -85,B 0,C 180,E1 -14741.177,E2 -14741.177} C_VEL
LIN {X 0,Y 326.756,Z 277.392,A -85,B 0,C 180,E1 -14745.433,E2 -14745.433} C_VEL
LIN {X 0,Y 326.763,Z 277.405,A -85,B 0,C 180,E1 -14748.839,E2 -14748.839} C_VEL
LIN {X 0,Y 326.952,Z 277.373,A -85,B 0,C 180,E1 -14752.59,E2 -14752.59} C_VEL
LIN {X 0,Y 326.771,Z 277.403,A -85,B 0,C 180,E1 -14755.065,E2 -14755.065} C_VEL
LIN {X 0,Y 327.041,Z 277.35,A -85,B 0,C 180,E1 -14757.537,E2 -14757.537} C_VEL
LIN {X 0,Y 327.211,Z 277.348,A -85,B 0,C 180,E1 -14760,E2 -14760} C_VEL
LIN {X 0,Y 327.04,Z 277.363,A -85,B 0,C 180,E1 -14762.463,E2 -14762.463} C_VEL
LIN {X 0,Y 326.989,Z 277.374,A -85,B 0,C 180,E1 -14766.169,E2 -14766.169} C_VEL
LIN {X 0,Y 326.908,Z 277.381,A -85,B 0,C 180,E1 -14768.655,E2 -14768.655} C_VEL
LIN {X 0,Y 326.727,Z 277.408,A -85,B 0,C 180,E1 -14772.421,E2 -14772.421} C_VEL
LIN {X 0,Y 326.747,Z 277.402,A -85,B 0,C 180,E1 -14774.958,E2 -14774.958} C_VEL
LIN {X 0,Y 326.726,Z 277.411,A -85,B 0,C 180,E1 -14778.838,E2 -14778.838} C_VEL
LIN {X 0,Y 326.616,Z 277.414,A -85,B 0,C 180,E1 -14782.788,E2 -14782.788} C_VEL
LIN {X 0,Y 326.684,Z 277.417,A -85,B 0,C 180,E1 -14785.484,E2 -14785.484} C_VEL
LIN {X 0,Y 326.655,Z 277.421,A -85,B 0,C 180,E1 -14789.66,E2 -14789.66} C_VEL
LIN {X 0,Y 326.601,Z 277.38,A -85,B 0,C 180,E1 -14794.02,E2 -14794.02} C_VEL
LIN {X 0,Y 326.623,Z 277.417,A -85,B 0,C 180,E1 -14797.239,E2 -14797.239} C_VEL
LIN {X 0,Y 326.573,Z 277.423,A -85,B 0,C 180,E1 -14801.132,E2 -14801.132} C_VEL
LIN {X 0,Y 326.581,Z 277.426,A -85,B 0,C 180,E1 -14804.754,E2 -14804.754} C_VEL
LIN {X 0,Y 326.618,Z 277.399,A -85,B 0,C 180,E1 -14808.162,E2 -14808.162} C_VEL
LIN {X 0,Y 326.644,Z 277.418,A -85,B 0,C 180,E1 -14811.395,E2 -14811.395} C_VEL
LIN {X 0,Y 326.665,Z 277.571,A -85,B 0,C 180,E1 -14815.102,E2 -14815.102} C_VEL
LIN {X 0,Y 329.45,Z 288.928,A -85,B 0,C 180,E1 -14818.573,E2 -14818.573} C_VEL
LIN {X 0,Y 330.601,Z 293.78,A -85,B 0,C 180,E1 -14819.927,E2 -14819.927} C_VEL
LIN {X 0,Y 334.911,Z 303.622,A -85,B 0,C 180,E1 -14820.635,E2 -14820.635} C_VEL
LIN {X 0,Y 339.281,Z 314.335,A -85,B 0,C 180,E1 -14821.302,E2 -14821.302} C_VEL
LIN {X 0,Y 343.067,Z 334.563,A -85,B 0,C 180,E1 -14822.118,E2 -14822.118} C_VEL
LIN {X 0,Y 340.799,Z 426.397,A -85,B 0,C 180,E1 -14824.051,E2 -14824.051} C_VEL
LIN {X 0,Y 339.986,Z 441.409,A -85,B 0,C 180,E1 -14824.519,E2 -14824.519} C_VEL
LIN {X 0,Y 338.847,Z 454.911,A -85,B 0,C 180,E1 -14825.166,E2 -14825.166} C_VEL
LIN {X 0,Y 337.453,Z 468.161,A -85,B 0,C 180,E1 -14826.039,E2 -14826.039} C_VEL
LIN {X 0,Y 335.846,Z 481.427,A -85,B 0,C 180,E1 -14827.185,E2 -14827.185} C_VEL
LIN {X 0,Y 334.047,Z 493.952,A -85,B 0,C 180,E1 -14828.559,E2 -14828.559} C_VEL
LIN {X 0,Y 332.395,Z 504.013,A -85,B 0,C 180,E1 -14829.905,E2 -14829.905} C_VEL
LIN {X 0,Y 330.551,Z 515.077,A -85,B 0,C 180,E1 -14831.724,E2 -14831.724} C_VEL
LIN {X 0,Y 329.014,Z 524.207,A -85,B 0,C 180,E1 -14833.559,E2 -14833.559} C_VEL
LIN {X 0,Y 327.583,Z 532.932,A -85,B 0,C 180,E1 -14835.717,E2 -14835.717} C_VEL
LIN {X 0,Y 326.606,Z 539.076,A -85,B 0,C 180,E1 -14837.574,E2 -14837.574} C_VEL
LIN {X 0,Y 325.676,Z 545.602,A -85,B 0,C 180,E1 -14840.059,E2 -14840.059} C_VEL
LIN {X 0,Y 325.173,Z 550.486,A -85,B 0,C 180,E1 -14842.549,E2 -14842.549} C_VEL
LIN {X 0,Y 324.89,Z 553.881,A -85,B 0,C 180,E1 -14845.036,E2 -14845.036} C_VEL
LIN {X 0,Y 324.802,Z 555.888,A -85,B 0,C 180,E1 -14847.52,E2 -14847.52} C_VEL
LIN {X 0,Y 324.791,Z 556.55,A -85,B 0,C 180,E1 -14850,E2 -14850} C_VEL
LIN {X 0,Y 324.802,Z 555.879,A -85,B 0,C 180,E1 -14852.48,E2 -14852.48} C_VEL
LIN {X 0,Y 324.892,Z 553.865,A -85,B 0,C 180,E1 -14854.964,E2 -14854.964} C_VEL
LIN {X 0,Y 325.173,Z 550.46,A -85,B 0,C 180,E1 -14857.451,E2 -14857.451} C_VEL
LIN {X 0,Y 325.679,Z 545.56,A -85,B 0,C 180,E1 -14859.941,E2 -14859.941} C_VEL
LIN {X 0,Y 326.606,Z 539.023,A -85,B 0,C 180,E1 -14862.426,E2 -14862.426} C_VEL
LIN {X 0,Y 327.586,Z 532.868,A -85,B 0,C 180,E1 -14864.283,E2 -14864.283} C_VEL
LIN {X 0,Y 328.746,Z 525.482,A -85,B 0,C 180,E1 -14866.136,E2 -14866.136} C_VEL
LIN {X 0,Y 330.235,Z 516.609,A -85,B 0,C 180,E1 -14867.974,E2 -14867.974} C_VEL
LIN {X 0,Y 332.026,Z 505.862,A -85,B 0,C 180,E1 -14869.796,E2 -14869.796} C_VEL
LIN {X 0,Y 333.882,Z 494.985,A -85,B 0,C 180,E1 -14871.29,E2 -14871.29} C_VEL
LIN {X 0,Y 335.674,Z 482.613,A -85,B 0,C 180,E1 -14872.678,E2 -14872.678} C_VEL
LIN {X 0,Y 337.271,Z 469.883,A -85,B 0,C 180,E1 -14873.811,E2 -14873.811} C_VEL
LIN {X 0,Y 338.742,Z 455.874,A -85,B 0,C 180,E1 -14874.761,E2 -14874.761} C_VEL
LIN {X 0,Y 339.89,Z 441.855,A -85,B 0,C 180,E1 -14875.448,E2 -14875.448} C_VEL
LIN {X 0,Y 340.679,Z 428.648,A -85,B 0,C 180,E1 -14875.876,E2 -14875.876} C_VEL
LIN {X 0,Y 343.11,Z 335.645,A -85,B 0,C 180,E1 -14877.833,E2 -14877.833} C_VEL
LIN {X 0,Y 339.229,Z 314.177,A -85,B 0,C 180,E1 -14878.684,E2 -14878.684} C_VEL
LIN {X 0,Y 333.368,Z 300.124,A -85,B 0,C 180,E1 -14879.574,E2 -14879.574} C_VEL
LIN {X 0,Y 330.649,Z 293.906,A -85,B 0,C 180,E1 -14880.029,E2 -14880.029} C_VEL
LIN {X 0,Y 328.135,Z 283.509,A -85,B 0,C 180,E1 -14883.01,E2 -14883.01} C_VEL
LIN {X 0,Y 326.654,Z 277.474,A -85,B 0,C 180,E1 -14884.935,E2 -14884.935} C_VEL
LIN {X 0,Y 326.595,Z 277.425,A -85,B 0,C 180,E1 -14888.612,E2 -14888.612} C_VEL
LIN {X 0,Y 326.573,Z 277.405,A -85,B 0,C 180,E1 -14891.845,E2 -14891.845} C_VEL
LIN {X 0,Y 326.524,Z 277.433,A -85,B 0,C 180,E1 -14895.257,E2 -14895.257} C_VEL
LIN {X 0,Y 326.574,Z 277.422,A -85,B 0,C 180,E1 -14898.868,E2 -14898.868} C_VEL
LIN {X 0,Y 326.624,Z 277.415,A -85,B 0,C 180,E1 -14902.761,E2 -14902.761} C_VEL
LIN {X 0,Y 326.602,Z 277.38,A -85,B 0,C 180,E1 -14905.98,E2 -14905.98} C_VEL
LIN {X 0,Y 326.656,Z 277.42,A -85,B 0,C 180,E1 -14910.341,E2 -14910.341} C_VEL
LIN {X 0,Y 326.685,Z 277.417,A -85,B 0,C 180,E1 -14914.516,E2 -14914.516} C_VEL
LIN {X 0,Y 326.643,Z 277.411,A -85,B 0,C 180,E1 -14918.545,E2 -14918.545} C_VEL
LIN {X 0,Y 326.739,Z 277.409,A -85,B 0,C 180,E1 -14921.177,E2 -14921.177} C_VEL
LIN {X 0,Y 326.757,Z 277.403,A -85,B 0,C 180,E1 -14925.433,E2 -14925.433} C_VEL
LIN {X 0,Y 326.763,Z 277.394,A -85,B 0,C 180,E1 -14928.839,E2 -14928.839} C_VEL
LIN {X 0,Y 326.973,Z 277.379,A -85,B 0,C 180,E1 -14932.59,E2 -14932.59} C_VEL
LIN {X 0,Y 326.771,Z 277.392,A -85,B 0,C 180,E1 -14935.065,E2 -14935.065} C_VEL
LIN {X 0,Y 327.041,Z 277.363,A -85,B 0,C 180,E1 -14937.537,E2 -14937.537} C_VEL
LIN {X 0,Y 327.192,Z 277.35,A -85,B 0,C 180,E1 -14940,E2 -14940} C_VEL
LIN {X 0,Y 327.041,Z 277.35,A -85,B 0,C 180,E1 -14942.463,E2 -14942.463} C_VEL
LIN {X 0,Y 326.954,Z 277.376,A -85,B 0,C 180,E1 -14946.64,E2 -14946.64} C_VEL
LIN {X 0,Y 326.799,Z 277.39,A -85,B 0,C 180,E1 -14949.907,E2 -14949.907} C_VEL
LIN {X 0,Y 326.753,Z 277.398,A -85,B 0,C 180,E1 -14953.686,E2 -14953.686} C_VEL
LIN {X 0,Y 326.694,Z 277.417,A -85,B 0,C 180,E1 -14957.528,E2 -14957.528} C_VEL
LIN {X 0,Y 326.657,Z 277.409,A -85,B 0,C 180,E1 -14960.136,E2 -14960.136} C_VEL
LIN {X 0,Y 326.647,Z 277.42,A -85,B 0,C 180,E1 -14964.129,E2 -14964.129} C_VEL
LIN {X 0,Y 326.68,Z 277.405,A -85,B 0,C 180,E1 -14966.858,E2 -14966.858} C_VEL
LIN {X 0,Y 326.635,Z 277.41,A -85,B 0,C 180,E1 -14970.612,E2 -14970.612} C_VEL
LIN {X 0,Y 326.603,Z 277.379,A -85,B 0,C 180,E1 -14974.02,E2 -14974.02} C_VEL
LIN {X 0,Y 326.626,Z 277.425,A -85,B 0,C 180,E1 -14977.24,E2 -14977.24} C_VEL
LIN {X 0,Y 326.597,Z 277.4,A -85,B 0,C 180,E1 -14980.208,E2 -14980.208} C_VEL
LIN {X 0,Y 326.575,Z 277.416,A -85,B 0,C 180,E1 -14983.524,E2 -14983.524} C_VEL
LIN {X 0,Y 326.58,Z 277.407,A -85,B 0,C 180,E1 -14987.028,E2 -14987.028} C_VEL
LIN {X 0,Y 326.61,Z 277.423,A -85,B 0,C 180,E1 -14990.773,E2 -14990.773} C_VEL
LIN {X 0,Y 326.612,Z 277.426,A -85,B 0,C 180,E1 -14994.481,E2 -14994.481} C_VEL
LIN {X 0,Y 326.613,Z 277.511,A -85,B 0,C 180,E1 -14996.419,E2 -14996.419} C_VEL
LIN {X 0,Y 328.762,Z 285.953,A -85,B 0,C 180,E1 -14999.133,E2 -14999.133} C_VEL
LIN {X 0,Y 329.448,Z 288.795,A -85,B 0,C 180,E1 -14999.907,E2 -14999.907} C_VEL
LIN {X 0,Y 337.04,Z 305.707,A -85,B 0,C 180,E1 -15001.088,E2 -15001.088} C_VEL
LIN {X 0,Y 341.422,Z 316.977,A -85,B 0,C 180,E1 -15001.759,E2 -15001.759} C_VEL
LIN {X 0,Y 343.293,Z 326.915,A -85,B 0,C 180,E1 -15002.158,E2 -15002.158} C_VEL
LIN {X 0,Y 341.209,Z 407.417,A -85,B 0,C 180,E1 -15003.838,E2 -15003.838} C_VEL
LIN {X 0,Y 340.549,Z 427.905,A -85,B 0,C 180,E1 -15004.318,E2 -15004.318} C_VEL
LIN {X 0,Y 339.634,Z 441.756,A -85,B 0,C 180,E1 -15004.859,E2 -15004.859} C_VEL
LIN {X 0,Y 338.386,Z 455.536,A -85,B 0,C 180,E1 -15005.637,E2 -15005.637} C_VEL
LIN {X 0,Y 336.949,Z 468.915,A -85,B 0,C 180,E1 -15006.654,E2 -15006.654} C_VEL
LIN {X 0,Y 335.389,Z 481.137,A -85,B 0,C 180,E1 -15007.841,E2 -15007.841} C_VEL
LIN {X 0,Y 333.667,Z 492.336,A -85,B 0,C 180,E1 -15009.18,E2 -15009.18} C_VEL
LIN {X 0,Y 331.83,Z 503.594,A -85,B 0,C 180,E1 -15010.836,E2 -15010.836} C_VEL
LIN {X 0,Y 330.043,Z 513.651,A -85,B 0,C 180,E1 -15012.656,E2 -15012.656} C_VEL
LIN {X 0,Y 328.517,Z 522.91,A -85,B 0,C 180,E1 -15014.725,E2 -15014.725} C_VEL
LIN {X 0,Y 327.41,Z 529.972,A -85,B 0,C 180,E1 -15016.659,E2 -15016.659} C_VEL
LIN {X 0,Y 326.336,Z 536.391,A -85,B 0,C 180,E1 -15018.824,E2 -15018.824} C_VEL
LIN {X 0,Y 325.524,Z 542.082,A -85,B 0,C 180,E1 -15021.308,E2 -15021.308} C_VEL
LIN {X 0,Y 325.145,Z 546.331,A -85,B 0,C 180,E1 -15023.876,E2 -15023.876} C_VEL
LIN {X 0,Y 324.927,Z 548.921,A -85,B 0,C 180,E1 -15026.28,E2 -15026.28} C_VEL
LIN {X 0,Y 324.787,Z 550.276,A -85,B 0,C 180,E1 -15028.76,E2 -15028.76} C_VEL
LIN {X 0,Y 324.787,Z 550.308,A -85,B 0,C 180,E1 -15031.24,E2 -15031.24} C_VEL
LIN {X 0,Y 324.927,Z 549.014,A -85,B 0,C 180,E1 -15033.72,E2 -15033.72} C_VEL
LIN {X 0,Y 325.153,Z 546.366,A -85,B 0,C 180,E1 -15036.204,E2 -15036.204} C_VEL
LIN {X 0,Y 325.521,Z 542.294,A -85,B 0,C 180,E1 -15038.692,E2 -15038.692} C_VEL
LIN {X 0,Y 326.314,Z 536.669,A -85,B 0,C 180,E1 -15041.177,E2 -15041.177} C_VEL
LIN {X 0,Y 327.368,Z 530.317,A -85,B 0,C 180,E1 -15043.343,E2 -15043.343} C_VEL
LIN {X 0,Y 328.46,Z 523.344,A -85,B 0,C 180,E1 -15045.274,E2 -15045.274} C_VEL
LIN {X 0,Y 330.004,Z 514.157,A -85,B 0,C 180,E1 -15047.346,E2 -15047.346} C_VEL
LIN {X 0,Y 331.708,Z 504.201,A -85,B 0,C 180,E1 -15049.171,E2 -15049.171} C_VEL
LIN {X 0,Y 333.571,Z 493.117,A -85,B 0,C 180,E1 -15050.826,E2 -15050.826} C_VEL
LIN {X 0,Y 335.43,Z 480.915,A -85,B 0,C 180,E1 -15052.291,E2 -15052.291} C_VEL
LIN {X 0,Y 337.062,Z 468.523,A -85,B 0,C 180,E1 -15053.484,E2 -15053.484} C_VEL
LIN {X 0,Y 338.437,Z 455.719,A -85,B 0,C 180,E1 -15054.457,E2 -15054.457} C_VEL
LIN {X 0,Y 339.685,Z 441.541,A -85,B 0,C 180,E1 -15055.259,E2 -15055.259} C_VEL
LIN {X 0,Y 340.573,Z 427.566,A -85,B 0,C 180,E1 -15055.803,E2 -15055.803} C_VEL
LIN {X 0,Y 341.44,Z 403.296,A -85,B 0,C 180,E1 -15056.348,E2 -15056.348} C_VEL
LIN {X 0,Y 342.9,Z 343.245,A -85,B 0,C 180,E1 -15057.609,E2 -15057.609} C_VEL
LIN {X 0,Y 342.469,Z 337.418,A -85,B 0,C 180,E1 -15057.782,E2 -15057.782} C_VEL
LIN {X 0,Y 341.067,Z 331.82,A -85,B 0,C 180,E1 -15058.037,E2 -15058.037} C_VEL
LIN {X 0,Y 336.652,Z 321.196,A -85,B 0,C 180,E1 -15058.692,E2 -15058.692} C_VEL
LIN {X 0,Y 333.487,Z 314.193,A -85,B 0,C 180,E1 -15059.159,E2 -15059.159} C_VEL
LIN {X 0,Y 326.02,Z 296.927,A -85,B 0,C 180,E1 -15060.326,E2 -15060.326} C_VEL
LIN {X 0,Y 322.185,Z 288.707,A -85,B 0,C 180,E1 -15060.982,E2 -15060.982} C_VEL
LIN {X 0,Y 319.653,Z 278.79,A -85,B 0,C 180,E1 -15064.099,E2 -15064.099} C_VEL
LIN {X 0,Y 319.579,Z 278.294,A -85,B 0,C 180,E1 -15064.49,E2 -15064.49} C_VEL
LIN {X 0,Y 319.541,Z 278.292,A -85,B 0,C 180,E1 -15068.011,E2 -15068.011} C_VEL
LIN {X 0,Y 319.523,Z 278.289,A -85,B 0,C 180,E1 -15071.596,E2 -15071.596} C_VEL
LIN {X 0,Y 319.513,Z 278.312,A -85,B 0,C 180,E1 -15075.261,E2 -15075.261} C_VEL
LIN {X 0,Y 319.528,Z 278.271,A -85,B 0,C 180,E1 -15078.712,E2 -15078.712} C_VEL
LIN {X 0,Y 319.574,Z 278.306,A -85,B 0,C 180,E1 -15082.343,E2 -15082.343} C_VEL
LIN {X 0,Y 319.555,Z 278.272,A -85,B 0,C 180,E1 -15085.123,E2 -15085.123} C_VEL
LIN {X 0,Y 319.565,Z 278.285,A -85,B 0,C 180,E1 -15089.057,E2 -15089.057} C_VEL
LIN {X 0,Y 319.604,Z 278.296,A -85,B 0,C 180,E1 -15092.498,E2 -15092.498} C_VEL
LIN {X 0,Y 319.599,Z 278.295,A -85,B 0,C 180,E1 -15095.303,E2 -15095.303} C_VEL
LIN {X 0,Y 319.591,Z 278.294,A -85,B 0,C 180,E1 -15098.047,E2 -15098.047} C_VEL
LIN {X 0,Y 319.683,Z 278.284,A -85,B 0,C 180,E1 -15100.962,E2 -15100.962} C_VEL
LIN {X 0,Y 319.724,Z 278.267,A -85,B 0,C 180,E1 -15105.276,E2 -15105.276} C_VEL
LIN {X 0,Y 319.746,Z 278.273,A -85,B 0,C 180,E1 -15109.872,E2 -15109.872} C_VEL
LIN {X 0,Y 319.906,Z 278.248,A -85,B 0,C 180,E1 -15112.425,E2 -15112.425} C_VEL
LIN {X 0,Y 319.741,Z 278.28,A -85,B 0,C 180,E1 -15114.956,E2 -15114.956} C_VEL
LIN {X 0,Y 319.985,Z 278.229,A -85,B 0,C 180,E1 -15117.482,E2 -15117.482} C_VEL
LIN {X 0,Y 320.162,Z 278.226,A -85,B 0,C 180,E1 -15120,E2 -15120} C_VEL
LIN {X 0,Y 319.984,Z 278.241,A -85,B 0,C 180,E1 -15122.518,E2 -15122.518} C_VEL
LIN {X 0,Y 319.944,Z 278.252,A -85,B 0,C 180,E1 -15126.306,E2 -15126.306} C_VEL
LIN {X 0,Y 319.836,Z 278.26,A -85,B 0,C 180,E1 -15128.848,E2 -15128.848} C_VEL
LIN {X 0,Y 319.675,Z 278.291,A -85,B 0,C 180,E1 -15132.7,E2 -15132.7} C_VEL
LIN {X 0,Y 319.693,Z 278.279,A -85,B 0,C 180,E1 -15135.296,E2 -15135.296} C_VEL
LIN {X 0,Y 319.668,Z 278.29,A -85,B 0,C 180,E1 -15139.255,E2 -15139.255} C_VEL
LIN {X 0,Y 319.566,Z 278.296,A -85,B 0,C 180,E1 -15143.32,E2 -15143.32} C_VEL
LIN {X 0,Y 319.629,Z 278.289,A -85,B 0,C 180,E1 -15146.088,E2 -15146.088} C_VEL
LIN {X 0,Y 319.584,Z 278.299,A -85,B 0,C 180,E1 -15148.934,E2 -15148.934} C_VEL
LIN {X 0,Y 319.527,Z 278.292,A -85,B 0,C 180,E1 -15151.862,E2 -15151.862} C_VEL
LIN {X 0,Y 319.574,Z 278.261,A -85,B 0,C 180,E1 -15155.543,E2 -15155.543} C_VEL
LIN {X 0,Y 319.568,Z 278.302,A -85,B 0,C 180,E1 -15158.009,E2 -15158.009} C_VEL
LIN {X 0,Y 319.522,Z 278.305,A -85,B 0,C 180,E1 -15161.598,E2 -15161.598} C_VEL
LIN {X 0,Y 319.572,Z 278.302,A -85,B 0,C 180,E1 -15165.274,E2 -15165.274} C_VEL
LIN {X 0,Y 319.575,Z 278.276,A -85,B 0,C 180,E1 -15168.72,E2 -15168.72} C_VEL
LIN {X 0,Y 319.58,Z 278.285,A -85,B 0,C 180,E1 -15172.344,E2 -15172.344} C_VEL
LIN {X 0,Y 319.611,Z 278.529,A -85,B 0,C 180,E1 -15174.53,E2 -15174.53} C_VEL
LIN {X 0,Y 322.076,Z 288.52,A -85,B 0,C 180,E1 -15177.676,E2 -15177.676} C_VEL
LIN {X 0,Y 323.384,Z 293.852,A -85,B 0,C 180,E1 -15179.201,E2 -15179.201} C_VEL
LIN {X 0,Y 331.331,Z 311.689,A -85,B 0,C 180,E1 -15180.484,E2 -15180.484} C_VEL
LIN {X 0,Y 333.386,Z 317.122,A -85,B 0,C 180,E1 -15180.815,E2 -15180.815} C_VEL
LIN {X 0,Y 336.839,Z 335.859,A -85,B 0,C 180,E1 -15181.587,E2 -15181.587} C_VEL
LIN {X 0,Y 334.346,Z 427.853,A -85,B 0,C 180,E1 -15183.554,E2 -15183.554} C_VEL
LIN {X 0,Y 333.534,Z 442.269,A -85,B 0,C 180,E1 -15184.031,E2 -15184.031} C_VEL
LIN {X 0,Y 332.284,Z 456.153,A -85,B 0,C 180,E1 -15184.725,E2 -15184.725} C_VEL
LIN {X 0,Y 330.771,Z 470.053,A -85,B 0,C 180,E1 -15185.691,E2 -15185.691} C_VEL
LIN {X 0,Y 329.022,Z 483.351,A -85,B 0,C 180,E1 -15186.91,E2 -15186.91} C_VEL
LIN {X 0,Y 327.245,Z 495.064,A -85,B 0,C 180,E1 -15188.256,E2 -15188.256} C_VEL
LIN {X 0,Y 325.359,Z 505.916,A -85,B 0,C 180,E1 -15189.781,E2 -15189.781} C_VEL
LIN {X 0,Y 323.479,Z 516.642,A -85,B 0,C 180,E1 -15191.638,E2 -15191.638} C_VEL
LIN {X 0,Y 321.907,Z 525.497,A -85,B 0,C 180,E1 -15193.512,E2 -15193.512} C_VEL
LIN {X 0,Y 320.524,Z 533.985,A -85,B 0,C 180,E1 -15195.72,E2 -15195.72} C_VEL
LIN {X 0,Y 319.336,Z 540.824,A -85,B 0,C 180,E1 -15197.932,E2 -15197.932} C_VEL
LIN {X 0,Y 318.631,Z 545.536,A -85,B 0,C 180,E1 -15199.837,E2 -15199.837} C_VEL
LIN {X 0,Y 318.093,Z 550.42,A -85,B 0,C 180,E1 -15202.382,E2 -15202.382} C_VEL
LIN {X 0,Y 317.81,Z 553.815,A -85,B 0,C 180,E1 -15204.925,E2 -15204.925} C_VEL
LIN {X 0,Y 317.725,Z 555.822,A -85,B 0,C 180,E1 -15207.465,E2 -15207.465} C_VEL
LIN {X 0,Y 317.702,Z 556.484,A -85,B 0,C 180,E1 -15210,E2 -15210} C_VEL
LIN {X 0,Y 317.725,Z 555.812,A -85,B 0,C 180,E1 -15212.536,E2 -15212.536} C_VEL
LIN {X 0,Y 317.813,Z 553.798,A -85,B 0,C 180,E1 -15215.075,E2 -15215.075} C_VEL
LIN {X 0,Y 318.093,Z 550.392,A -85,B 0,C 180,E1 -15217.618,E2 -15217.618} C_VEL
LIN {X 0,Y 318.634,Z 545.492,A -85,B 0,C 180,E1 -15220.163,E2 -15220.163} C_VEL
LIN {X 0,Y 319.337,Z 540.768,A -85,B 0,C 180,E1 -15222.068,E2 -15222.068} C_VEL
LIN {X 0,Y 320.524,Z 533.918,A -85,B 0,C 180,E1 -15224.281,E2 -15224.281} C_VEL
LIN {X 0,Y 321.878,Z 525.413,A -85,B 0,C 180,E1 -15226.49,E2 -15226.49} C_VEL
LIN {X 0,Y 323.464,Z 516.54,A -85,B 0,C 180,E1 -15228.363,E2 -15228.363} C_VEL
LIN {X 0,Y 325.313,Z 505.792,A -85,B 0,C 180,E1 -15230.222,E2 -15230.222} C_VEL
LIN {X 0,Y 327.273,Z 494.915,A -85,B 0,C 180,E1 -15231.742,E2 -15231.742} C_VEL
LIN {X 0,Y 329.168,Z 482.104,A -85,B 0,C 180,E1 -15233.203,E2 -15233.203} C_VEL
LIN {X 0,Y 330.779,Z 469.811,A -85,B 0,C 180,E1 -15234.308,E2 -15234.308} C_VEL
LIN {X 0,Y 332.32,Z 455.8,A -85,B 0,C 180,E1 -15235.272,E2 -15235.272} C_VEL
LIN {X 0,Y 333.492,Z 441.778,A -85,B 0,C 180,E1 -15235.972,E2 -15235.972} C_VEL
LIN {X 0,Y 334.323,Z 428.565,A -85,B 0,C 180,E1 -15236.406,E2 -15236.406} C_VEL
LIN {X 0,Y 336.707,Z 340.107,A -85,B 0,C 180,E1 -15238.301,E2 -15238.301} C_VEL
LIN {X 0,Y 336.646,Z 335.039,A -85,B 0,C 180,E1 -15238.427,E2 -15238.427} C_VEL
LIN {X 0,Y 333.049,Z 316.011,A -85,B 0,C 180,E1 -15239.221,E2 -15239.221} C_VEL
LIN {X 0,Y 326.449,Z 300.675,A -85,B 0,C 180,E1 -15240.25,E2 -15240.25} C_VEL
LIN {X 0,Y 323.362,Z 293.733,A -85,B 0,C 180,E1 -15240.789,E2 -15240.789} C_VEL
LIN {X 0,Y 320.984,Z 283.958,A -85,B 0,C 180,E1 -15243.694,E2 -15243.694} C_VEL
LIN {X 0,Y 319.581,Z 278.355,A -85,B 0,C 180,E1 -15245.543,E2 -15245.543} C_VEL
LIN {X 0,Y 319.556,Z 278.3,A -85,B 0,C 180,E1 -15249.668,E2 -15249.668} C_VEL
LIN {X 0,Y 319.519,Z 278.304,A -85,B 0,C 180,E1 -15253.46,E2 -15253.46} C_VEL
LIN {X 0,Y 319.55,Z 278.306,A -85,B 0,C 180,E1 -15257.016,E2 -15257.016} C_VEL
LIN {X 0,Y 319.543,Z 278.302,A -85,B 0,C 180,E1 -15260.37,E2 -15260.37} C_VEL
LIN {X 0,Y 319.554,Z 278.277,A -85,B 0,C 180,E1 -15263.572,E2 -15263.572} C_VEL
LIN {X 0,Y 319.573,Z 278.262,A -85,B 0,C 180,E1 -15266.686,E2 -15266.686} C_VEL
LIN {X 0,Y 319.587,Z 278.3,A -85,B 0,C 180,E1 -15269.616,E2 -15269.616} C_VEL
LIN {X 0,Y 319.604,Z 278.285,A -85,B 0,C 180,E1 -15272.498,E2 -15272.498} C_VEL
LIN {X 0,Y 319.601,Z 278.299,A -85,B 0,C 180,E1 -15275.304,E2 -15275.304} C_VEL
LIN {X 0,Y 319.592,Z 278.286,A -85,B 0,C 180,E1 -15278.047,E2 -15278.047} C_VEL
LIN {X 0,Y 319.683,Z 278.288,A -85,B 0,C 180,E1 -15280.962,E2 -15280.962} C_VEL
LIN {X 0,Y 319.725,Z 278.278,A -85,B 0,C 180,E1 -15285.276,E2 -15285.276} C_VEL
LIN {X 0,Y 319.751,Z 278.263,A -85,B 0,C 180,E1 -15289.873,E2 -15289.873} C_VEL
LIN {X 0,Y 319.927,Z 278.257,A -85,B 0,C 180,E1 -15292.426,E2 -15292.426} C_VEL
LIN {X 0,Y 319.74,Z 278.268,A -85,B 0,C 180,E1 -15294.956,E2 -15294.956} C_VEL
LIN {X 0,Y 319.985,Z 278.241,A -85,B 0,C 180,E1 -15297.482,E2 -15297.482} C_VEL
LIN {X 0,Y 320.143,Z 278.228,A -85,B 0,C 180,E1 -15300,E2 -15300} C_VEL
LIN {X 0,Y 319.985,Z 278.229,A -85,B 0,C 180,E1 -15302.518,E2 -15302.518} C_VEL
LIN {X 0,Y 319.915,Z 278.253,A -85,B 0,C 180,E1 -15306.628,E2 -15306.628} C_VEL
LIN {X 0,Y 319.746,Z 278.271,A -85,B 0,C 180,E1 -15310.128,E2 -15310.128} C_VEL
LIN {X 0,Y 319.725,Z 278.267,A -85,B 0,C 180,E1 -15314.724,E2 -15314.724} C_VEL
LIN {X 0,Y 319.684,Z 278.285,A -85,B 0,C 180,E1 -15319.038,E2 -15319.038} C_VEL
LIN {X 0,Y 319.565,Z 278.306,A -85,B 0,C 180,E1 -15323.32,E2 -15323.32} C_VEL
LIN {X 0,Y 319.63,Z 278.281,A -85,B 0,C 180,E1 -15326.089,E2 -15326.089} C_VEL
LIN {X 0,Y 319.586,Z 278.304,A -85,B 0,C 180,E1 -15328.934,E2 -15328.934} C_VEL
LIN {X 0,Y 319.528,Z 278.273,A -85,B 0,C 180,E1 -15331.862,E2 -15331.862} C_VEL
LIN {X 0,Y 319.576,Z 278.276,A -85,B 0,C 180,E1 -15335.544,E2 -15335.544} C_VEL
LIN {X 0,Y 319.578,Z 278.302,A -85,B 0,C 180,E1 -15338.008,E2 -15338.008} C_VEL
LIN {X 0,Y 319.526,Z 278.27,A -85,B 0,C 180,E1 -15341.598,E2 -15341.598} C_VEL
LIN {X 0,Y 319.514,Z 278.309,A -85,B 0,C 180,E1 -15345.263,E2 -15345.263} C_VEL
LIN {X 0,Y 319.526,Z 278.289,A -85,B 0,C 180,E1 -15348.712,E2 -15348.712} C_VEL
LIN {X 0,Y 319.553,Z 278.289,A -85,B 0,C 180,E1 -15352.35,E2 -15352.35} C_VEL
LIN {X 0,Y 319.607,Z 278.496,A -85,B 0,C 180,E1 -15355.895,E2 -15355.895} C_VEL
LIN {X 0,Y 322.185,Z 288.655,A -85,B 0,C 180,E1 -15359.127,E2 -15359.127} C_VEL
LIN {X 0,Y 325.544,Z 295.972,A -85,B 0,C 180,E1 -15359.717,E2 -15359.717} C_VEL
LIN {X 0,Y 332.015,Z 310.618,A -85,B 0,C 180,E1 -15360.726,E2 -15360.726} C_VEL
LIN {X 0,Y 335.407,Z 319.492,A -85,B 0,C 180,E1 -15361.264,E2 -15361.264} C_VEL
LIN {X 0,Y 337.021,Z 328.744,A -85,B 0,C 180,E1 -15361.635,E2 -15361.635} C_VEL
LIN {X 0,Y 334.789,Z 409.297,A -85,B 0,C 180,E1 -15363.34,E2 -15363.34} C_VEL
LIN {X 0,Y 334.086,Z 429.126,A -85,B 0,C 180,E1 -15363.826,E2 -15363.826} C_VEL
LIN {X 0,Y 333.157,Z 442.595,A -85,B 0,C 180,E1 -15364.377,E2 -15364.377} C_VEL
LIN {X 0,Y 331.928,Z 455.61,A -85,B 0,C 180,E1 -15365.131,E2 -15365.131} C_VEL
LIN {X 0,Y 330.427,Z 468.988,A -85,B 0,C 180,E1 -15366.165,E2 -15366.165} C_VEL
LIN {X 0,Y 328.825,Z 481.209,A -85,B 0,C 180,E1 -15367.374,E2 -15367.374} C_VEL
LIN {X 0,Y 326.856,Z 493.532,A -85,B 0,C 180,E1 -15368.891,E2 -15368.891} C_VEL
LIN {X 0,Y 325.098,Z 503.664,A -85,B 0,C 180,E1 -15370.423,E2 -15370.423} C_VEL
LIN {X 0,Y 323.255,Z 513.72,A -85,B 0,C 180,E1 -15372.28,E2 -15372.28} C_VEL
LIN {X 0,Y 321.808,Z 521.904,A -85,B 0,C 180,E1 -15374.115,E2 -15374.115} C_VEL
LIN {X 0,Y 320.671,Z 529.033,A -85,B 0,C 180,E1 -15376.05,E2 -15376.05} C_VEL
LIN {X 0,Y 319.574,Z 534.783,A -85,B 0,C 180,E1 -15377.941,E2 -15377.941} C_VEL
LIN {X 0,Y 318.875,Z 539.508,A -85,B 0,C 180,E1 -15379.845,E2 -15379.845} C_VEL
LIN {X 0,Y 318.232,Z 544.403,A -85,B 0,C 180,E1 -15382.386,E2 -15382.386} C_VEL
LIN {X 0,Y 317.915,Z 547.809,A -85,B 0,C 180,E1 -15384.927,E2 -15384.927} C_VEL
LIN {X 0,Y 317.762,Z 549.831,A -85,B 0,C 180,E1 -15387.465,E2 -15387.465} C_VEL
LIN {X 0,Y 317.704,Z 550.524,A -85,B 0,C 180,E1 -15390,E2 -15390} C_VEL
LIN {X 0,Y 317.761,Z 549.894,A -85,B 0,C 180,E1 -15392.535,E2 -15392.535} C_VEL
LIN {X 0,Y 317.915,Z 547.928,A -85,B 0,C 180,E1 -15395.073,E2 -15395.073} C_VEL
LIN {X 0,Y 318.232,Z 544.581,A -85,B 0,C 180,E1 -15397.614,E2 -15397.614} C_VEL
LIN {X 0,Y 318.848,Z 539.752,A -85,B 0,C 180,E1 -15400.156,E2 -15400.156} C_VEL
LIN {X 0,Y 319.546,Z 535.091,A -85,B 0,C 180,E1 -15402.06,E2 -15402.06} C_VEL
LIN {X 0,Y 320.821,Z 528.312,A -85,B 0,C 180,E1 -15404.267,E2 -15404.267} C_VEL
LIN {X 0,Y 321.981,Z 521.165,A -85,B 0,C 180,E1 -15406.177,E2 -15406.177} C_VEL
LIN {X 0,Y 323.487,Z 512.724,A -85,B 0,C 180,E1 -15408.034,E2 -15408.034} C_VEL
LIN {X 0,Y 325.324,Z 502.401,A -85,B 0,C 180,E1 -15409.891,E2 -15409.891} C_VEL
LIN {X 0,Y 327.374,Z 490.851,A -85,B 0,C 180,E1 -15411.569,E2 -15411.569} C_VEL
LIN {X 0,Y 329.214,Z 478.848,A -85,B 0,C 180,E1 -15412.983,E2 -15412.983} C_VEL
LIN {X 0,Y 330.746,Z 466.641,A -85,B 0,C 180,E1 -15414.144,E2 -15414.144} C_VEL
LIN {X 0,Y 332.227,Z 453.52,A -85,B 0,C 180,E1 -15415.112,E2 -15415.112} C_VEL
LIN {X 0,Y 333.474,Z 439.312,A -85,B 0,C 180,E1 -15415.89,E2 -15415.89} C_VEL
LIN {X 0,Y 334.341,Z 425.306,A -85,B 0,C 180,E1 -15416.404,E2 -15416.404} C_VEL
LIN {X 0,Y 336.454,Z 351.305,A -85,B 0,C 180,E1 -15417.995,E2 -15417.995} C_VEL
LIN {X 0,Y 336.939,Z 327.343,A -85,B 0,C 180,E1 -15418.519,E2 -15418.519} C_VEL
LIN {X 0,Y 335.114,Z 318.162,A -85,B 0,C 180,E1 -15418.909,E2 -15418.909} C_VEL
LIN {X 0,Y 333.487,Z 314.193,A -85,B 0,C 180,E1 -15419.159,E2 -15419.159} C_VEL
LIN {X 0,Y 330.833,Z 309.394,A -85,B 0,C 180,E1 -15419.534,E2 -15419.534} C_VEL
LIN {X 0,Y 325.093,Z 302.56,A -85,B 0,C 180,E1 -15420.281,E2 -15420.281} C_VEL
LIN {X 0,Y 318.045,Z 294.498,A -85,B 0,C 180,E1 -15421.235,E2 -15421.235} C_VEL
LIN {X 0,Y 316.105,Z 291.431,A -85,B 0,C 180,E1 -15421.529,E2 -15421.529} C_VEL
LIN {X 0,Y 314.908,Z 288.556,A -85,B 0,C 180,E1 -15421.816,E2 -15421.816} C_VEL
LIN {X 0,Y 312.54,Z 279.334,A -85,B 0,C 180,E1 -15424.889,E2 -15424.889} C_VEL
LIN {X 0,Y 312.491,Z 279.17,A -85,B 0,C 180,E1 -15428.079,E2 -15428.079} C_VEL
LIN {X 0,Y 312.487,Z 279.178,A -85,B 0,C 180,E1 -15430.708,E2 -15430.708} C_VEL
LIN {X 0,Y 312.47,Z 279.179,A -85,B 0,C 180,E1 -15434.205,E2 -15434.205} C_VEL
LIN {X 0,Y 312.485,Z 279.15,A -85,B 0,C 180,E1 -15437.917,E2 -15437.917} C_VEL
LIN {X 0,Y 312.532,Z 279.184,A -85,B 0,C 180,E1 -15441.909,E2 -15441.909} C_VEL
LIN {X 0,Y 312.501,Z 279.139,A -85,B 0,C 180,E1 -15445.789,E2 -15445.789} C_VEL
LIN {X 0,Y 312.519,Z 279.16,A -85,B 0,C 180,E1 -15448.853,E2 -15448.853} C_VEL
LIN {X 0,Y 312.57,Z 279.175,A -85,B 0,C 180,E1 -15451.824,E2 -15451.824} C_VEL
LIN {X 0,Y 312.58,Z 279.162,A -85,B 0,C 180,E1 -15454.71,E2 -15454.71} C_VEL
LIN {X 0,Y 312.582,Z 279.169,A -85,B 0,C 180,E1 -15457.528,E2 -15457.528} C_VEL
LIN {X 0,Y 312.632,Z 279.166,A -85,B 0,C 180,E1 -15461.656,E2 -15461.656} C_VEL
LIN {X 0,Y 312.687,Z 279.145,A -85,B 0,C 180,E1 -15465.686,E2 -15465.686} C_VEL
LIN {X 0,Y 312.692,Z 279.152,A -85,B 0,C 180,E1 -15469.641,E2 -15469.641} C_VEL
LIN {X 0,Y 312.847,Z 279.126,A -85,B 0,C 180,E1 -15472.254,E2 -15472.254} C_VEL
LIN {X 0,Y 312.71,Z 279.157,A -85,B 0,C 180,E1 -15474.842,E2 -15474.842} C_VEL
LIN {X 0,Y 312.986,Z 279.108,A -85,B 0,C 180,E1 -15478.713,E2 -15478.713} C_VEL
LIN {X 0,Y 313.114,Z 279.103,A -85,B 0,C 180,E1 -15480,E2 -15480} C_VEL
LIN {X 0,Y 312.93,Z 279.119,A -85,B 0,C 180,E1 -15482.574,E2 -15482.574} C_VEL
LIN {X 0,Y 312.903,Z 279.131,A -85,B 0,C 180,E1 -15486.448,E2 -15486.448} C_VEL
LIN {X 0,Y 312.781,Z 279.138,A -85,B 0,C 180,E1 -15489.049,E2 -15489.049} C_VEL
LIN {X 0,Y 312.627,Z 279.167,A -85,B 0,C 180,E1 -15492.991,E2 -15492.991} C_VEL
LIN {X 0,Y 312.631,Z 279.154,A -85,B 0,C 180,E1 -15495.65,E2 -15495.65} C_VEL
LIN {X 0,Y 312.624,Z 279.167,A -85,B 0,C 180,E1 -15499.237,E2 -15499.237} C_VEL
LIN {X 0,Y 312.54,Z 279.166,A -85,B 0,C 180,E1 -15502.79,E2 -15502.79} C_VEL
LIN {X 0,Y 312.597,Z 279.167,A -85,B 0,C 180,E1 -15505.936,E2 -15505.936} C_VEL
LIN {X 0,Y 312.54,Z 279.179,A -85,B 0,C 180,E1 -15509.65,E2 -15509.65} C_VEL
LIN {X 0,Y 312.514,Z 279.135,A -85,B 0,C 180,E1 -15513.689,E2 -15513.689} C_VEL
LIN {X 0,Y 312.521,Z 279.174,A -85,B 0,C 180,E1 -15517.386,E2 -15517.386} C_VEL
LIN {X 0,Y 312.486,Z 279.175,A -85,B 0,C 180,E1 -15520.71,E2 -15520.71} C_VEL
LIN {X 0,Y 312.506,Z 279.176,A -85,B 0,C 180,E1 -15524.2,E2 -15524.2} C_VEL
LIN {X 0,Y 312.545,Z 279.152,A -85,B 0,C 180,E1 -15527.906,E2 -15527.906} C_VEL
LIN {X 0,Y 312.542,Z 279.165,A -85,B 0,C 180,E1 -15531.909,E2 -15531.909} C_VEL
LIN {X 0,Y 312.553,Z 279.394,A -85,B 0,C 180,E1 -15533.883,E2 -15533.883} C_VEL
LIN {X 0,Y 314.855,Z 288.474,A -85,B 0,C 180,E1 -15536.848,E2 -15536.848} C_VEL
LIN {X 0,Y 316.138,Z 293.68,A -85,B 0,C 180,E1 -15538.403,E2 -15538.403} C_VEL
LIN {X 0,Y 324.858,Z 313.02,A -85,B 0,C 180,E1 -15539.87,E2 -15539.87} C_VEL
LIN {X 0,Y 327.594,Z 320.29,A -85,B 0,C 180,E1 -15540.327,E2 -15540.327} C_VEL
LIN {X 0,Y 330.591,Z 337.149,A -85,B 0,C 180,E1 -15541.032,E2 -15541.032} C_VEL
LIN {X 0,Y 327.955,Z 429.309,A -85,B 0,C 180,E1 -15543.04,E2 -15543.04} C_VEL
LIN {X 0,Y 327.014,Z 444.028,A -85,B 0,C 180,E1 -15543.56,E2 -15543.56} C_VEL
LIN {X 0,Y 325.754,Z 457.356,A -85,B 0,C 180,E1 -15544.267,E2 -15544.267} C_VEL
LIN {X 0,Y 324.301,Z 469.992,A -85,B 0,C 180,E1 -15545.174,E2 -15545.174} C_VEL
LIN {X 0,Y 322.512,Z 483.063,A -85,B 0,C 180,E1 -15546.39,E2 -15546.39} C_VEL
LIN {X 0,Y 320.637,Z 495,A -85,B 0,C 180,E1 -15547.785,E2 -15547.785} C_VEL
LIN {X 0,Y 318.658,Z 505.852,A -85,B 0,C 180,E1 -15549.337,E2 -15549.337} C_VEL
LIN {X 0,Y 316.726,Z 516.577,A -85,B 0,C 180,E1 -15551.232,E2 -15551.232} C_VEL
LIN {X 0,Y 315.062,Z 525.432,A -85,B 0,C 180,E1 -15553.143,E2 -15553.143} C_VEL
LIN {X 0,Y 313.578,Z 533.92,A -85,B 0,C 180,E1 -15555.396,E2 -15555.396} C_VEL
LIN {X 0,Y 312.35,Z 540.758,A -85,B 0,C 180,E1 -15557.658,E2 -15557.658} C_VEL
LIN {X 0,Y 311.604,Z 545.47,A -85,B 0,C 180,E1 -15559.605,E2 -15559.605} C_VEL
LIN {X 0,Y 311.027,Z 550.354,A -85,B 0,C 180,E1 -15562.208,E2 -15562.208} C_VEL
LIN {X 0,Y 310.718,Z 553.749,A -85,B 0,C 180,E1 -15564.809,E2 -15564.809} C_VEL
LIN {X 0,Y 310.649,Z 555.756,A -85,B 0,C 180,E1 -15567.407,E2 -15567.407} C_VEL
LIN {X 0,Y 310.616,Z 556.417,A -85,B 0,C 180,E1 -15570,E2 -15570} C_VEL
LIN {X 0,Y 310.65,Z 555.746,A -85,B 0,C 180,E1 -15572.593,E2 -15572.593} C_VEL
LIN {X 0,Y 310.722,Z 553.731,A -85,B 0,C 180,E1 -15575.191,E2 -15575.191} C_VEL
LIN {X 0,Y 311.027,Z 550.324,A -85,B 0,C 180,E1 -15577.792,E2 -15577.792} C_VEL
LIN {X 0,Y 311.607,Z 545.424,A -85,B 0,C 180,E1 -15580.395,E2 -15580.395} C_VEL
LIN {X 0,Y 312.681,Z 538.887,A -85,B 0,C 180,E1 -15582.989,E2 -15582.989} C_VEL
LIN {X 0,Y 313.952,Z 531.613,A -85,B 0,C 180,E1 -15585.25,E2 -15585.25} C_VEL
LIN {X 0,Y 315.555,Z 522.601,A -85,B 0,C 180,E1 -15587.498,E2 -15587.498} C_VEL
LIN {X 0,Y 317.323,Z 513.147,A -85,B 0,C 180,E1 -15589.403,E2 -15589.403} C_VEL
LIN {X 0,Y 319.223,Z 502.679,A -85,B 0,C 180,E1 -15591.131,E2 -15591.131} C_VEL
LIN {X 0,Y 321.259,Z 491.127,A -85,B 0,C 180,E1 -15592.679,E2 -15592.679} C_VEL
LIN {X 0,Y 323.14,Z 478.392,A -85,B 0,C 180,E1 -15594.057,E2 -15594.057} C_VEL
LIN {X 0,Y 324.778,Z 465.776,A -85,B 0,C 180,E1 -15595.129,E2 -15595.129} C_VEL
LIN {X 0,Y 326.328,Z 451.824,A -85,B 0,C 180,E1 -15596.027,E2 -15596.027} C_VEL
LIN {X 0,Y 327.401,Z 438.041,A -85,B 0,C 180,E1 -15596.665,E2 -15596.665} C_VEL
LIN {X 0,Y 328.163,Z 423.891,A -85,B 0,C 180,E1 -15597.07,E2 -15597.07} C_VEL
LIN {X 0,Y 330.549,Z 337.492,A -85,B 0,C 180,E1 -15598.939,E2 -15598.939} C_VEL
LIN {X 0,Y 327.184,Z 318.881,A -85,B 0,C 180,E1 -15599.724,E2 -15599.724} C_VEL
LIN {X 0,Y 321.1,Z 304.535,A -85,B 0,C 180,E1 -15600.708,E2 -15600.708} C_VEL
LIN {X 0,Y 316.157,Z 293.74,A -85,B 0,C 180,E1 -15601.559,E2 -15601.559} C_VEL
LIN {X 0,Y 313.857,Z 284.35,A -85,B 0,C 180,E1 -15604.429,E2 -15604.429} C_VEL
LIN {X 0,Y 312.519,Z 279.223,A -85,B 0,C 180,E1 -15606.194,E2 -15606.194} C_VEL
LIN {X 0,Y 312.501,Z 279.169,A -85,B 0,C 180,E1 -15610.125,E2 -15610.125} C_VEL
LIN {X 0,Y 312.455,Z 279.189,A -85,B 0,C 180,E1 -15613.965,E2 -15613.965} C_VEL
LIN {X 0,Y 312.48,Z 279.187,A -85,B 0,C 180,E1 -15617.918,E2 -15617.918} C_VEL
LIN {X 0,Y 312.531,Z 279.179,A -85,B 0,C 180,E1 -15621.91,E2 -15621.91} C_VEL
LIN {X 0,Y 312.501,Z 279.133,A -85,B 0,C 180,E1 -15625.789,E2 -15625.789} C_VEL
LIN {X 0,Y 312.519,Z 279.177,A -85,B 0,C 180,E1 -15628.853,E2 -15628.853} C_VEL
LIN {X 0,Y 312.57,Z 279.164,A -85,B 0,C 180,E1 -15631.824,E2 -15631.824} C_VEL
LIN {X 0,Y 312.581,Z 279.173,A -85,B 0,C 180,E1 -15634.711,E2 -15634.711} C_VEL
LIN {X 0,Y 312.582,Z 279.158,A -85,B 0,C 180,E1 -15637.529,E2 -15637.529} C_VEL
LIN {X 0,Y 312.632,Z 279.163,A -85,B 0,C 180,E1 -15641.656,E2 -15641.656} C_VEL
LIN {X 0,Y 312.688,Z 279.158,A -85,B 0,C 180,E1 -15645.686,E2 -15645.686} C_VEL
LIN {X 0,Y 312.696,Z 279.141,A -85,B 0,C 180,E1 -15649.642,E2 -15649.642} C_VEL
LIN {X 0,Y 312.865,Z 279.137,A -85,B 0,C 180,E1 -15652.254,E2 -15652.254} C_VEL
LIN {X 0,Y 312.711,Z 279.145,A -85,B 0,C 180,E1 -15654.842,E2 -15654.842} C_VEL
LIN {X 0,Y 312.984,Z 279.121,A -85,B 0,C 180,E1 -15658.713,E2 -15658.713} C_VEL
LIN {X 0,Y 312.984,Z 279.108,A -85,B 0,C 180,E1 -15661.287,E2 -15661.287} C_VEL
LIN {X 0,Y 312.711,Z 279.156,A -85,B 0,C 180,E1 -15665.158,E2 -15665.158} C_VEL
LIN {X 0,Y 312.847,Z 279.126,A -85,B 0,C 180,E1 -15667.746,E2 -15667.746} C_VEL
LIN {X 0,Y 312.663,Z 279.164,A -85,B 0,C 180,E1 -15671.672,E2 -15671.672} C_VEL
LIN {X 0,Y 312.694,Z 279.142,A -85,B 0,C 180,E1 -15674.888,E2 -15674.888} C_VEL
LIN {X 0,Y 312.625,Z 279.162,A -85,B 0,C 180,E1 -15679.237,E2 -15679.237} C_VEL
LIN {X 0,Y 312.541,Z 279.175,A -85,B 0,C 180,E1 -15682.79,E2 -15682.79} C_VEL
LIN {X 0,Y 312.598,Z 279.157,A -85,B 0,C 180,E1 -15685.936,E2 -15685.936} C_VEL
LIN {X 0,Y 312.542,Z 279.175,A -85,B 0,C 180,E1 -15689.651,E2 -15689.651} C_VEL
LIN {X 0,Y 312.516,Z 279.13,A -85,B 0,C 180,E1 -15693.689,E2 -15693.689} C_VEL
LIN {X 0,Y 312.537,Z 279.18,A -85,B 0,C 180,E1 -15697.384,E2 -15697.384} C_VEL
LIN {X 0,Y 312.49,Z 279.149,A -85,B 0,C 180,E1 -15700.709,E2 -15700.709} C_VEL
LIN {X 0,Y 312.471,Z 279.184,A -85,B 0,C 180,E1 -15704.206,E2 -15704.206} C_VEL
LIN {X 0,Y 312.484,Z 279.16,A -85,B 0,C 180,E1 -15707.919,E2 -15707.919} C_VEL
LIN {X 0,Y 312.497,Z 279.178,A -85,B 0,C 180,E1 -15710.972,E2 -15710.972} C_VEL
LIN {X 0,Y 312.531,Z 279.177,A -85,B 0,C 180,E1 -15715.011,E2 -15715.011} C_VEL
LIN {X 0,Y 312.636,Z 279.729,A -85,B 0,C 180,E1 -15715.417,E2 -15715.417} C_VEL
LIN {X 0,Y 314.912,Z 288.675,A -85,B 0,C 180,E1 -15718.32,E2 -15718.32} C_VEL
LIN {X 0,Y 317.154,Z 293.5,A -85,B 0,C 180,E1 -15718.76,E2 -15718.76} C_VEL
LIN {X 0,Y 324.994,Z 310.557,A -85,B 0,C 180,E1 -15720.025,E2 -15720.025} C_VEL
LIN {X 0,Y 329.429,Z 321.928,A -85,B 0,C 180,E1 -15720.75,E2 -15720.75} C_VEL
LIN {X 0,Y 330.772,Z 329.658,A -85,B 0,C 180,E1 -15721.069,E2 -15721.069} C_VEL
LIN {X 0,Y 328.48,Z 409.388,A -85,B 0,C 180,E1 -15722.786,E2 -15722.786} C_VEL
LIN {X 0,Y 327.744,Z 429.208,A -85,B 0,C 180,E1 -15723.28,E2 -15723.28} C_VEL
LIN {X 0,Y 326.787,Z 442.671,A -85,B 0,C 180,E1 -15723.84,E2 -15723.84} C_VEL
LIN {X 0,Y 325.42,Z 456.588,A -85,B 0,C 180,E1 -15724.667,E2 -15724.667} C_VEL
LIN {X 0,Y 323.872,Z 469.56,A -85,B 0,C 180,E1 -15725.7,E2 -15725.7} C_VEL
LIN {X 0,Y 322.078,Z 482.643,A -85,B 0,C 180,E1 -15727.043,E2 -15727.043} C_VEL
LIN {X 0,Y 320.044,Z 494.67,A -85,B 0,C 180,E1 -15728.588,E2 -15728.588} C_VEL
LIN {X 0,Y 318.092,Z 505.512,A -85,B 0,C 180,E1 -15730.31,E2 -15730.31} C_VEL
LIN {X 0,Y 316.171,Z 515.272,A -85,B 0,C 180,E1 -15732.204,E2 -15732.204} C_VEL
LIN {X 0,Y 314.669,Z 523.529,A -85,B 0,C 180,E1 -15734.166,E2 -15734.166} C_VEL
LIN {X 0,Y 313.549,Z 530.109,A -85,B 0,C 180,E1 -15736.057,E2 -15736.057} C_VEL
LIN {X 0,Y 312.337,Z 536.527,A -85,B 0,C 180,E1 -15738.316,E2 -15738.316} C_VEL
LIN {X 0,Y 311.452,Z 542.217,A -85,B 0,C 180,E1 -15740.912,E2 -15740.912} C_VEL
LIN {X 0,Y 310.988,Z 546.351,A -85,B 0,C 180,E1 -15743.512,E2 -15743.512} C_VEL
LIN {X 0,Y 310.754,Z 549.055,A -85,B 0,C 180,E1 -15746.11,E2 -15746.11} C_VEL
LIN {X 0,Y 310.618,Z 550.409,A -85,B 0,C 180,E1 -15748.703,E2 -15748.703} C_VEL
LIN {X 0,Y 310.618,Z 550.441,A -85,B 0,C 180,E1 -15751.296,E2 -15751.296} C_VEL
LIN {X 0,Y 310.754,Z 549.147,A -85,B 0,C 180,E1 -15753.89,E2 -15753.89} C_VEL
LIN {X 0,Y 310.988,Z 546.498,A -85,B 0,C 180,E1 -15756.488,E2 -15756.488} C_VEL
LIN {X 0,Y 311.442,Z 542.426,A -85,B 0,C 180,E1 -15759.088,E2 -15759.088} C_VEL
LIN {X 0,Y 312.313,Z 536.8,A -85,B 0,C 180,E1 -15761.684,E2 -15761.684} C_VEL
LIN {X 0,Y 313.493,Z 530.447,A -85,B 0,C 180,E1 -15763.945,E2 -15763.945} C_VEL
LIN {X 0,Y 314.851,Z 522.894,A -85,B 0,C 180,E1 -15766.108,E2 -15766.108} C_VEL
LIN {X 0,Y 316.431,Z 514.285,A -85,B 0,C 180,E1 -15768.116,E2 -15768.116} C_VEL
LIN {X 0,Y 318.282,Z 504.328,A -85,B 0,C 180,E1 -15770.014,E2 -15770.014} C_VEL
LIN {X 0,Y 320.318,Z 493.242,A -85,B 0,C 180,E1 -15771.73,E2 -15771.73} C_VEL
LIN {X 0,Y 322.162,Z 482.204,A -85,B 0,C 180,E1 -15773.12,E2 -15773.12} C_VEL
LIN {X 0,Y 323.89,Z 470.218,A -85,B 0,C 180,E1 -15774.347,E2 -15774.347} C_VEL
LIN {X 0,Y 325.451,Z 456.964,A -85,B 0,C 180,E1 -15775.416,E2 -15775.416} C_VEL
LIN {X 0,Y 326.725,Z 443.939,A -85,B 0,C 180,E1 -15776.208,E2 -15776.208} C_VEL
LIN {X 0,Y 327.75,Z 429.948,A -85,B 0,C 180,E1 -15776.806,E2 -15776.806} C_VEL
LIN {X 0,Y 328.433,Z 412.323,A -85,B 0,C 180,E1 -15777.261,E2 -15777.261} C_VEL
LIN {X 0,Y 330.324,Z 346.679,A -85,B 0,C 180,E1 -15778.675,E2 -15778.675} C_VEL
LIN {X 0,Y 330.665,Z 328.076,A -85,B 0,C 180,E1 -15779.094,E2 -15779.094} C_VEL
LIN {X 0,Y 329.048,Z 320.547,A -85,B 0,C 180,E1 -15779.436,E2 -15779.436} C_VEL
LIN {X 0,Y 321.622,Z 302.901,A -85,B 0,C 180,E1 -15780.635,E2 -15780.635} C_VEL
LIN {X 0,Y 316.105,Z 291.431,A -85,B 0,C 180,E1 -15781.529,E2 -15781.529} C_VEL
LIN {X 0,Y 314.422,Z 289.353,A -85,B 0,C 180,E1 -15781.834,E2 -15781.834} C_VEL
LIN {X 0,Y 311.72,Z 287.66,A -85,B 0,C 180,E1 -15782.43,E2 -15782.43} C_VEL
LIN {X 0,Y 308.834,Z 286.119,A -85,B 0,C 180,E1 -15783.246,E2 -15783.246} C_VEL
LIN {X 0,Y 306.706,Z 284.05,A -85,B 0,C 180,E1 -15784.147,E2 -15784.147} C_VEL
LIN {X 0,Y 306.149,Z 282.788,A -85,B 0,C 180,E1 -15784.61,E2 -15784.61} C_VEL
LIN {X 0,Y 305.488,Z 280.09,A -85,B 0,C 180,E1 -15785.665,E2 -15785.665} C_VEL
LIN {X 0,Y 305.438,Z 280.05,A -85,B 0,C 180,E1 -15788.526,E2 -15788.526} C_VEL
LIN {X 0,Y 305.456,Z 280.035,A -85,B 0,C 180,E1 -15792.586,E2 -15792.586} C_VEL
LIN {X 0,Y 305.441,Z 280.052,A -85,B 0,C 180,E1 -15796.347,E2 -15796.347} C_VEL
LIN {X 0,Y 305.456,Z 280.032,A -85,B 0,C 180,E1 -15799.892,E2 -15799.892} C_VEL
LIN {X 0,Y 305.495,Z 280.052,A -85,B 0,C 180,E1 -15803.626,E2 -15803.626} C_VEL
LIN {X 0,Y 305.46,Z 280.011,A -85,B 0,C 180,E1 -15806.482,E2 -15806.482} C_VEL
LIN {X 0,Y 305.491,Z 280.059,A -85,B 0,C 180,E1 -15810.949,E2 -15810.949} C_VEL
LIN {X 0,Y 305.566,Z 280.032,A -85,B 0,C 180,E1 -15814.087,E2 -15814.087} C_VEL
LIN {X 0,Y 305.494,Z 280.044,A -85,B 0,C 180,E1 -15818.402,E2 -15818.402} C_VEL
LIN {X 0,Y 305.584,Z 280.043,A -85,B 0,C 180,E1 -15821.217,E2 -15821.217} C_VEL
LIN {X 0,Y 305.642,Z 280.02,A -85,B 0,C 180,E1 -15825.349,E2 -15825.349} C_VEL
LIN {X 0,Y 305.629,Z 280.033,A -85,B 0,C 180,E1 -15829.399,E2 -15829.399} C_VEL
LIN {X 0,Y 305.79,Z 280.004,A -85,B 0,C 180,E1 -15832.074,E2 -15832.074} C_VEL
LIN {X 0,Y 305.681,Z 280.033,A -85,B 0,C 180,E1 -15834.723,E2 -15834.723} C_VEL
LIN {X 0,Y 305.952,Z 279.983,A -85,B 0,C 180,E1 -15838.684,E2 -15838.684} C_VEL
LIN {X 0,Y 305.952,Z 279.997,A -85,B 0,C 180,E1 -15841.316,E2 -15841.316} C_VEL
LIN {X 0,Y 305.845,Z 280.012,A -85,B 0,C 180,E1 -15846.597,E2 -15846.597} C_VEL
LIN {X 0,Y 305.729,Z 280.015,A -85,B 0,C 180,E1 -15849.26,E2 -15849.26} C_VEL
LIN {X 0,Y 305.582,Z 280.044,A -85,B 0,C 180,E1 -15853.296,E2 -15853.296} C_VEL
LIN {X 0,Y 305.587,Z 280.028,A -85,B 0,C 180,E1 -15856.02,E2 -15856.02} C_VEL
LIN {X 0,Y 305.571,Z 280.046,A -85,B 0,C 180,E1 -15859.445,E2 -15859.445} C_VEL
LIN {X 0,Y 305.485,Z 280.046,A -85,B 0,C 180,E1 -15863.042,E2 -15863.042} C_VEL
LIN {X 0,Y 305.542,Z 280.042,A -85,B 0,C 180,E1 -15866.227,E2 -15866.227} C_VEL
LIN {X 0,Y 305.491,Z 280.054,A -85,B 0,C 180,E1 -15869.05,E2 -15869.05} C_VEL
LIN {X 0,Y 305.439,Z 280.044,A -85,B 0,C 180,E1 -15871.953,E2 -15871.953} C_VEL
LIN {X 0,Y 305.457,Z 280.013,A -85,B 0,C 180,E1 -15875.114,E2 -15875.114} C_VEL
LIN {X 0,Y 305.462,Z 280.061,A -85,B 0,C 180,E1 -15878.533,E2 -15878.533} C_VEL
LIN {X 0,Y 305.459,Z 280.061,A -85,B 0,C 180,E1 -15882.588,E2 -15882.588} C_VEL
LIN {X 0,Y 305.489,Z 280.052,A -85,B 0,C 180,E1 -15886.358,E2 -15886.358} C_VEL
LIN {X 0,Y 305.496,Z 280.042,A -85,B 0,C 180,E1 -15889.9,E2 -15889.9} C_VEL
LIN {X 0,Y 305.521,Z 280.178,A -85,B 0,C 180,E1 -15893.165,E2 -15893.165} C_VEL
LIN {X 0,Y 307.965,Z 289.874,A -85,B 0,C 180,E1 -15896.44,E2 -15896.44} C_VEL
LIN {X 0,Y 308.9,Z 293.711,A -85,B 0,C 180,E1 -15897.585,E2 -15897.585} C_VEL
LIN {X 0,Y 316.514,Z 310.097,A -85,B 0,C 180,E1 -15898.915,E2 -15898.915} C_VEL
LIN {X 0,Y 321.573,Z 322.308,A -85,B 0,C 180,E1 -15899.766,E2 -15899.766} C_VEL
LIN {X 0,Y 324.356,Z 338.693,A -85,B 0,C 180,E1 -15900.461,E2 -15900.461} C_VEL
LIN {X 0,Y 321.648,Z 429.26,A -85,B 0,C 180,E1 -15902.467,E2 -15902.467} C_VEL
